  IF fb_RFTrigManualMove.FT THEN
    mManuellMove( bI_Do                  := FALSE
                , fI_TargetPosition      := (fB_Axis.fO_ActualPosition * 1000)
                , fL_ManualMoveTolerance := fB_Axis.fI_Tolerance);
  END_IF
END_IF
(*Rest command if move is done*)
IF bL_Ready OR bL_Error THEN
  sADS_CleanAxis.ResetCommands();
END_IF

sL_CleanDevStatus := sStatus;

(*ADS Feedback*)
sADS_CleanAxis.setFeedback( bManualMoveCanEx := sADS_CleanAxis.bO_ManualMoveCanEx        // do not change
                          , bManualMovekExec := sADS_CleanAxis.bO_ManualMovekExec        // do not change
                          , fAxisPositionVal := fB_Axis.fO_ActualPosition * 1000
                          , wErrorCode       := wL_ErrorCode
                          , bBusy            := sL_CleanDevStatus.bBusy
                          , bReady           := sL_CleanDevStatus.bReady
                          , bError           := sL_CleanDevStatus.bError
                          );


(*----------------------------------------------------------------------------------------------------------------------------------------------- *)
(* Supervision  *)
(*----------------------------------------------------------------------------------------------------------------------------------------------- *)
(*
TODO: Supervisor
tL_TimerSurv.PT := T#3S;
tL_TimerSurv();
tL_TimerSensor.PT := T#105s  ;  (* 1meter at 10mm*)
tL_TimerSensor();*)

IF bL_FirstRun THEN
  bL_FirstRun     := FALSE;
END_IF;

(*----------------------------------------------------------------------------------------------------------------------- *)
(*--------------------------------- Fault Diagnosis and Management  ----------------------------------------------------- *)
(*----------------------------------------------------------------------------------------------------------------------- *)
mErrorHandling();

(*----------------------------------------------------------------------------------------------------------------------- *)
(* Messaging                                                                                                              *)
(*----------------------------------------------------------------------------------------------------------------------- *)
fB_MsgHandler();
fB_Msg[1](bI_Status := bL_Error);
fB_MsgQueue();

METHOD mAckError 
VAR_INPUT
END_VAR
wL_ErrorCode := 0;
mErrorHandling();
fB_Axis.bI_FaultReset := TRUE;
END_METHOD

METHOD mCapping : BOOL
VAR_INPUT
  iI_Step    : INT;
  bI_ExitCap : BOOL;
END_VAR
//Abort: Stop whereever axis is and return
IF bL_AbortReq THEN
  fB_Axis.bI_MoveEnable := FALSE;
  bL_Busy  := FALSE;
  bL_Ready := TRUE;

  RETURN;
END_IF

//Normal operation
bL_Ready := FALSE;
CASE iI_Step OF
	0: //Init - Check if axis is not activated, restore safety
    fB_Axis.bI_MoveEnable := FALSE;
		bL_Busy               := FALSE;

  1: //Wait for PU axis to lift
    mAckError();
    fB_Axis.fI_TargetPosition := (fI_PositionClean1 / 1000);
    fB_Axis.fI_SpeedLimit     := sI_SpeedDef.fP_PlaceSpeed / 1000;
    
    IF bL_InPosClean1 THEN
      fB_Axis.bI_MoveEnable := FALSE;
      bL_Busy               := FALSE;
      bL_Ready              := TRUE;  //Operation complete
    ELSE
      fB_Axis.bI_MoveEnable := bL_SafeMovePos;
      bL_Busy               := TRUE;
    END_IF
    
  2: //Wait for CU axis to move in
    fB_Axis.bI_MoveEnable   := FALSE;
    bL_Busy                 := FALSE;
    
  3: //Move CH to park positiom 
    fB_Axis.bI_MoveEnable   := FALSE;
    bL_Busy                 := FALSE;
    
  4: //Wait for PU axis to lower
    mAckError();
    IF NOT bI_ExitCap THEN
      fB_Axis.fI_TargetPosition := (fI_PositionClean2 / 1000);
      fB_Axis.fI_SpeedLimit     := sI_SpeedDef.fP_PlaceSpeed / 1000;
      
      IF bL_InPosClean2 THEN
        fB_Axis.bI_MoveEnable := FALSE;
        bL_Busy               := FALSE;
        bL_Ready              := TRUE;  //Operation complete
      ELSE
        fB_Axis.bI_MoveEnable := bL_SafeMoveNeg;
        bL_Busy               := TRUE;
      END_IF
    ELSE
      fB_Axis.bI_MoveEnable := FALSE;
      bL_Busy               := FALSE;
    END_IF
    
	5: //End - Do nothing, capping process active
    mAckError();
		bL_Busy  := FALSE;
    bL_Ready := TRUE;  //Operation complete

	ELSE
		bL_Busy  := FALSE;		
    bL_Ready := TRUE;  //Operation complete
END_CASE
END_METHOD

METHOD mCleaning : BOOL
VAR_INPUT
  iI_Step : INT;
END_VAR
//Abort: Stop whereever axis is and return
IF bL_AbortReq THEN
  fB_Axis.bI_MoveEnable := FALSE;
  bL_Busy  := FALSE;
  bL_Ready := TRUE;

  RETURN;
END_IF

//Normal operation
bL_Ready := FALSE;
CASE iI_Step OF
  0: //Init - Check if axis is not activated, restore safety
    bL_Busy := FALSE;

  1: //Wait for PU axis to lift
    mAckError();
    fB_Axis.fI_TargetPosition := (fI_PositionClean1 / 1000);
    fB_Axis.fI_SpeedLimit     := sI_SpeedDef.fP_PlaceSpeed / 1000;
    
    IF bL_InPosClean1 THEN
      fB_Axis.bI_MoveEnable := FALSE;
      bL_Busy               := FALSE;
      bL_Ready              := TRUE;  //Operation complete
    ELSE
      fB_Axis.bI_MoveEnable := bL_SafeMovePos;
      bL_Busy               := TRUE;
    END_IF
    
  2: //Wait for CU axis to move in
    fB_Axis.bI_MoveEnable   := FALSE;
    bL_Busy                 := FALSE;
    
  3: //Wait for PU axis to lower
    mAckError();
    fB_Axis.fI_TargetPosition := (fI_PositionClean2 / 1000);
    fB_Axis.fI_SpeedLimit     := sI_SpeedDef.fP_PlaceSpeed / 1000;
    
    IF bL_InPosClean2 THEN
      fB_Axis.bI_MoveEnable := FALSE;
      bL_Busy               := FALSE;
      bL_Ready              := TRUE;  //Operation complete
    ELSE
      fB_Axis.bI_MoveEnable := bL_SafeMoveNeg;
      bL_Busy               := TRUE;
    END_IF
    
  4: //Ensure CH axis is at starting position
    fB_Axis.bI_MoveEnable   := FALSE;
    bL_Busy                 := FALSE;
    
  5: //Move CH to clean start position
    fB_Axis.bI_MoveEnable   := FALSE;
    bL_Busy                 := FALSE;

  6: //Wait until cleaning equipment ready
    fB_Axis.bI_MoveEnable   := FALSE;
    bL_Busy                 := FALSE;
    
  7: //Cleaning
    fB_Axis.bI_MoveEnable   := FALSE;
    bL_Busy                 := FALSE;  
    
  8: //Wait until cleaning equipment ready
    fB_Axis.bI_MoveEnable   := FALSE;
    bL_Busy                 := FALSE;
    
  9: //Move CH to end position
    fB_Axis.bI_MoveEnable   := FALSE;
    bL_Busy                 := FALSE;  
    
  10: //Wait for PU axis to lift
    mAckError();
    fB_Axis.fI_TargetPosition := (fI_PositionClean1 / 1000);
    fB_Axis.fI_SpeedLimit     := sI_SpeedDef.fP_PlaceSpeed / 1000;
    
    IF bL_InPosClean1 THEN
      fB_Axis.bI_MoveEnable := FALSE;
      bL_Busy               := FALSE;
      bL_Ready              := TRUE;  //Operation complete
    ELSE
      fB_Axis.bI_MoveEnable := bL_SafeMovePos;
      bL_Busy               := TRUE;
    END_IF
  
  11: //Move CH back to start 
    fB_Axis.bI_MoveEnable   := FALSE;
    bL_Busy                 := FALSE;  

  12: //Wait for PU axis to lower
    mAckError();
    fB_Axis.fI_TargetPosition := (fI_PositionClean2 / 1000);
    fB_Axis.fI_SpeedLimit     := sI_SpeedDef.fP_PlaceSpeed / 1000;
    
    IF bL_InPosClean2 THEN
      fB_Axis.bI_MoveEnable := FALSE;
      bL_Busy               := FALSE;
      bL_Ready              := TRUE;  //Operation complete
    ELSE
      fB_Axis.bI_MoveEnable := bL_SafeMoveNeg;
      bL_Busy               := TRUE;
    END_IF
    
  13: //End
    fB_Axis.bI_MoveEnable   := FALSE;
    bL_Busy                 := FALSE;  
    bL_Ready                := TRUE;  //Operation complete
  
  ELSE
    bL_Busy  := FALSE;    
    bL_Ready := TRUE;  //Operation complete
END_CASE
END_METHOD

METHOD PRIVATE mErrorHandling
VAR_INPUT
END_VAR
fB_Msg[1].bI_Status := FALSE;

IF NOT bL_RefKnown THEN
	wL_ErrorCode.1 := TRUE;						(* Axis has lost its value *)
END_IF;

IF (NOT bI_SensorTop AND NOT bI_SensorBottom) THEN      (* Sensor Fault : SensorTop and SensorBottom can't be active at the same time *)
	wL_ErrorCode.2 := TRUE;
END_IF;

IF (NOT bI_SensorTop AND bL_MemSensorTop) THEN          (* Safety Fault : Limit Switch Top activated *)
	wL_ErrorCode.3 := TRUE;
END_IF;
bL_MemSensorTop := bI_SensorTop;

IF (NOT bI_SensorBottom AND bL_MemSensorBottom) THEN    (* Safety Fault : Limit Switch Bottom activated *)
	wL_ErrorCode.4 := TRUE;
END_IF;
bL_MemSensorBottom := bI_SensorBottom;

IF (sI_SpeedDef.fP_PlaceSpeed=0) OR  (sI_SpeedDef.fP_WorkSpeed=0) OR (sI_SpeedDef.fP_ServiceSpeed=0) THEN	(* Speed Configuration not done *)
	wL_Errorcode.6 := TRUE;
END_IF;

IF (fI_PositionService = 0) OR (fI_PositionWait = 0) OR (fI_PositionClean1 = 0) OR (fI_PositionClean2 = 0) THEN		(* Position Configuration not done *)
	wL_ErrorCode.7 := TRUE;
END_IF;

IF fB_Axis.eO_EL7201Status = eFault  THEN
	wL_ErrorCode.8 := TRUE;						(* EL7342 module fault *)
	fB_Msg[1].bI_Status := TRUE;
END_IF;


IF wl_ErrorCode = 0 THEN
	bL_Error := FALSE;
ELSE
	bL_Error := TRUE;
END_IF;
END_METHOD

METHOD mErrorRecovery : BOOL
VAR_INPUT
    iI_Step : INT;
END_VAR
//Do nothing
bL_Busy  := FALSE;
bL_Ready := TRUE;
END_METHOD

METHOD mInit
VAR_INPUT
END_VAR
	(*Messages*)
	sL_MsgConfig.bI_Enable       := TRUE;
	sL_MsgConfig.pI_FbMsgHandler := ADR(fB_MsgHandler);
	fB_MsgHandler.pI_MsgQueue    := ADR(fB_MsgQueue);
	fB_MsgQueue.pI_MsgInterface  := ADR(sADS_CleanAxis.sO_Message);
	fB_MsgQueue.cI_MaxElement    := 5;

	fB_Msg[1].iI_MsgLocation     := TO_INT(eMa_BLK_CLEANAXIS);
	fB_Msg[1].pI_MsgConfig       := ADR(sL_MsgConfig);
	fB_Msg[1].iI_MsgNumber       := eCMa_AxisErrorZ;
END_METHOD

METHOD mManuellMove : BOOL
VAR_INPUT
  bI_Do                  : BOOL;
  fI_TargetPosition      : REAL;
  fL_ManualMoveTolerance : REAL;
END_VAR
IF fB_Axis.fO_ActualPosition < (fI_PositionWait / 1000) THEN
  fB_Axis.fI_SpeedLimit   := sI_SpeedDef.fP_WorkSpeed / 1000;
ELSE
  fB_Axis.fI_SpeedLimit   := sI_SpeedDef.fP_ServiceSpeed / 1000;
END_IF
fB_Axis.fI_TargetPosition := fI_TargetPosition / 1000;
IF fB_Axis.fI_TargetPosition > fB_Axis.fO_ActualPosition THEN
  fB_Axis.bI_MoveEnable   := bI_Do AND bL_SafeMovePos;
ELSIF fB_Axis.fI_TargetPosition < fB_Axis.fO_ActualPosition THEN
  fB_Axis.bI_MoveEnable   := bI_Do AND bL_SafeMoveNeg;
ELSE
  fB_Axis.bI_MoveEnable   := bI_Do;
END_IF

bL_Busy  := ABS(fB_Axis.fI_TargetPosition - fB_Axis.fO_ActualPosition) > fL_ManualMoveTolerance;
bL_Ready := NOT (ABS(fB_Axis.fI_TargetPosition - fB_Axis.fO_ActualPosition) > fL_ManualMoveTolerance);  //Operation complete
END_METHOD

METHOD mPrintPos : BOOL
VAR_INPUT
  bI_PrintEnabled        : BOOL;
  bI_PrintFinsihed       : BOOL;
END_VAR

VAR
  bDriveToWaitPos        : BOOL;
  bDriveToPrintPos       : BOOL;
END_VAR
fb_RFTrigPrintEnabled(CLK := bI_PrintEnabled);
IF fb_RFTrigPrintEnabled.RT THEN bL_DriveToPrintPos := TRUE; bL_DriveToWaitPos  := FALSE; END_IF
IF fb_RFTrigPrintEnabled.FT THEN bL_DriveToWaitPos  := TRUE; bL_DriveToPrintPos := FALSE; END_IF

IF NOT pHigherPosWait AND bL_Ready THEN
  //IF fb_RFTrigPrintEnabled.RT THEN bL_DriveToPrintPos := TRUE; END_IF
  IF bL_DriveToPrintPos THEN
    fB_Axis.fI_TargetPosition := (fL_PrintPosition);
    fB_Axis.fI_SpeedLimit     := sI_SpeedDef.fP_WorkSpeed / 1000;
    
    IF bL_InPosPrint THEN
      fB_Axis.bI_MoveEnable := FALSE;
      bL_Busy               := FALSE;
      bL_DriveToPrintPos    := FALSE;
      bL_Ready              := TRUE;  //Operation complete
    ELSE
      fB_Axis.bI_MoveEnable := bL_SafeMoveNeg;
      bL_Busy               := TRUE;
    END_IF
  END_IF

  //IF fb_RFTrigPrintEnabled.FT THEN bL_bDriveToWaitPos := TRUE; END_IF
  IF bL_DriveToWaitPos AND bI_PrintFinsihed THEN
    fB_Axis.fI_TargetPosition := (fI_PositionWait / 1000);
    fB_Axis.fI_SpeedLimit     := sI_SpeedDef.fP_PlaceSpeed / 1000;
    
    IF bL_InPosWait THEN
      fB_Axis.bI_MoveEnable := FALSE;
      bL_Busy               := FALSE;
      bL_DriveToWaitPos     := FALSE;
      bL_Ready              := TRUE;  //Operation complete
    ELSE
      fB_Axis.bI_MoveEnable := bL_SafeMovePos;
      bL_Busy               := TRUE;
    END_IF
  END_IF
END_IF
END_METHOD

METHOD mProduction : BOOL
VAR_INPUT
  iI_Step : INT;
END_VAR
//Abort: Stop whereever axis is and return
IF bL_AbortReq THEN
  fB_Axis.bI_MoveEnable := FALSE;
  bL_Busy  := FALSE;
  bL_Ready := TRUE;

  RETURN;
END_IF

//Normal operation
bL_Ready := FALSE;
CASE iI_Step OF
  0: //Init - Check if axis is not activated, restore safety
    bL_Busy := FALSE;

  1: //Wait for PU axis to lift
    mAckError();
    fB_Axis.fI_TargetPosition := (fI_PositionClean1 / 1000);
    fB_Axis.fI_SpeedLimit     := sI_SpeedDef.fP_PlaceSpeed / 1000;
    
    IF bL_InPosClean1 THEN
      fB_Axis.bI_MoveEnable := FALSE;
      bL_Busy               := FALSE;
      bL_Ready              := TRUE;  //Operation complete
    ELSE
      fB_Axis.bI_MoveEnable := bL_SafeMovePos;
      bL_Busy               := TRUE;
    END_IF
    
  2: //Wait for CU axis to move out
    fB_Axis.bI_MoveEnable   := FALSE;
    bL_Busy                 := FALSE;
    
  3: //Wait for PU axis to lower
    mAckError();
    fB_Axis.fI_TargetPosition := (fI_PositionWait / 1000);
    fB_Axis.fI_SpeedLimit     := sI_SpeedDef.fP_PlaceSpeed / 1000;
    
    IF bL_InPosWait THEN
      fB_Axis.bI_MoveEnable := FALSE;
      bL_Busy               := FALSE;
      bL_Ready              := TRUE;  //Operation complete
    ELSE
      fB_Axis.bI_MoveEnable := bL_SafeMoveNeg;
      bL_Busy               := TRUE;
    END_IF
    
  4: //End
    fB_Axis.bI_MoveEnable := FALSE;
    bL_Busy               := FALSE;  
    bL_Ready              := TRUE;  //Operation complete

  ELSE
    bL_Busy  := FALSE;    
    bL_Ready := TRUE;  //Operation complete
END_CASE
END_METHOD

METHOD mService : BOOL
VAR_INPUT
  iI_Step : INT;
END_VAR
//Abort: Stop whereever axis is and return
IF bL_AbortReq THEN
  fB_Axis.bI_MoveEnable := FALSE;
  bL_Busy  := FALSE;
  bL_Ready := TRUE;

  RETURN;
END_IF

//Normal operation
bL_Ready := FALSE;
CASE iI_Step OF
  0: //Init - Check if axis is not activated, restore safety
    bL_Busy := FALSE;

  1: //Wait for PU axis to lift to ExitCapping
    mAckError();
    fB_Axis.fI_TargetPosition := (fI_PositionClean1 / 1000);
    fB_Axis.fI_SpeedLimit     := sI_SpeedDef.fP_PlaceSpeed / 1000;
    
    IF bL_InPosClean1 THEN
      fB_Axis.bI_MoveEnable := FALSE;
      bL_Busy               := FALSE;
    ELSE
      fB_Axis.bI_MoveEnable := bL_SafeMovePos;
      bL_Busy               := TRUE;
    END_IF
        
  2: //Wait for PU to reach Service (CU moves out)
    mAckError();
    fB_Axis.fI_TargetPosition := (fI_PositionService / 1000);
    fB_Axis.fI_SpeedLimit     := sI_SpeedDef.fP_PlaceSpeed / 1000;
    
    IF bL_InPosService THEN
      fB_Axis.bI_MoveEnable := FALSE;
      bL_Busy               := FALSE;
      bL_Ready              := TRUE;  //Operation complete
    ELSE
      fB_Axis.bI_MoveEnable := bL_SafeMovePos;
      bL_Busy               := TRUE;
    END_IF
    
  3: //End
    fB_Axis.bI_MoveEnable := FALSE;
    bL_Busy               := FALSE; 
    bL_Ready              := TRUE; 
  
  ELSE
    bL_Busy  := FALSE;    
    bL_Ready := TRUE;  //Operation complete
END_CASE
END_METHOD

METHOD mStartup : BOOL
VAR_INPUT
  iI_Step : INT;
END_VAR
CASE iI_Step OF
	0: //Init - Check if axis is not activated, restore safety
		bL_Busy := FALSE;

  1: //Wait for PU axis to lift
    mAckError();
    fB_Axis.fI_TargetPosition := (fI_PositionClean1 / 1000);
    fB_Axis.fI_SpeedLimit     := sI_SpeedDef.fP_PlaceSpeed / 1000;
    
    IF bL_InPosClean1 OR bL_HigherPosC1 THEN
      fB_Axis.bI_MoveEnable := FALSE;
      bL_Busy               := FALSE;
      bL_Ready              := TRUE;  //Operation complete
    ELSE
      fB_Axis.bI_MoveEnable := bL_SafeMovePos;
      bL_Busy               := TRUE;
    END_IF
    
	2,3,4: //End
		bL_Busy  := FALSE;		
    bL_Ready := TRUE;  //Operation complete

	ELSE
		bL_Busy  := FALSE;		
    bL_Ready := TRUE;  //Operation complete
END_CASE
END_METHOD

{attribute 'monitoring' := 'call'}
PROPERTY pHigherPosC1 : bool
GET
pHigherPosC1 := bL_HigherPosC1;
END_GET
END_PROPERTY

{attribute 'monitoring' := 'call'}
PROPERTY pHigherPosWait : bool
GET
pHigherPosWait := bL_HigherPosWait;
END_GET
END_PROPERTY

{attribute 'monitoring' := 'call'}
PROPERTY pInPosClean1 : bool
GET
pInPosClean1 := bL_InPosClean1;
END_GET
END_PROPERTY

{attribute 'monitoring' := 'call'}
PROPERTY pInPosClean2 : bool
GET
pInPosClean2 := bL_InPosClean2;
END_GET
END_PROPERTY

{attribute 'monitoring' := 'call'}
PROPERTY pInPosPrint : bool
GET
pInPosPrint := bL_InPosPrint;
END_GET
END_PROPERTY

{attribute 'monitoring' := 'call'}
PROPERTY pInPosService : bool
GET
pInPosService := bL_InPosService;
END_GET
END_PROPERTY

{attribute 'monitoring' := 'call'}
PROPERTY pInPosWait : bool
GET
pInPosWait := bL_InPosWait;
END_GET
END_PROPERTY

PROPERTY pPositionPrint : REAL
GET
pPositionPrint := fI_PositionPrint;
END_GET
SET
fI_PositionPrint := pPositionPrint;
END_SET
END_PROPERTY

PROPERTY setPlaceSpeed : REAL
SET
sI_SpeedDef.fP_PlaceSpeed := setPlaceSpeed;
END_SET
END_PROPERTY

END_FUNCTION_BLOCK

// ---- POUs/Machine/CleaningStation/FB_CleaningProcess.TcPOU
FUNCTION_BLOCK FB_CleaningProcess EXTENDS FB_MachineBase IMPLEMENTS I_CleaningStateCallback
VAR_INPUT
  I_CleanDeviceList              : ARRAY[1..cI_MAXCLEANDEVICES] OF I_CleanDevice;

  (*User commands*)
  bI_UsrService                  : BOOL;                         (*User has selected service (1) or print(0) mode*)
  bI_UsrAbort                    : BOOL;                         (*User aborted*)
  bI_Emergency                   : BOOL;
  bI_SafetyOk                    : BOOL;

  bI_CappingCommand              : BOOL;                         (*Capping command*)
  bI_PurgeCommand                : BOOL;                         (*Purge command*)
  bI_CleanCommand                : BOOL;                         (*Clean command*)
  bI_CleanLocked                 : BOOL;                         (*Cleaning locked*)
  
  (*User settings*)
  bI_UsrAutoMode                 : BOOL;                         (*User has selected automatic mode*)
  bI_UsrCleanAfterPurge          : BOOL;                         (*Automatically clean after Purge*)
  bI_UsrCleanAfterCapp           : BOOL;                         (*Automatically clean after Capping*)
  bI_UsrPurgeAfterCapp           : BOOL;                         (*Automatically purge after Capping*)

  bI_CappingPosReached           : BOOL;                         (*Capping position reached*)
  bI_CappingEnterPosReached      : BOOL;                         (*Capping enter position reached*)
END_VAR

VAR_OUTPUT
END_VAR

VAR
  sADS_CleanProcess              : FB_ADS_CleanProcess;

  fB_StateInit                   : FB_CleaningProcessStateInit;
  fB_StateProduction             : FB_CleaningProcessStateProduction;
  fB_StateService                : FB_CleaningProcessStateService;
  fB_StateCapping                : FB_CleaningProcessStateCapping;
  fB_StateCappingExit            : FB_CleaningProcessStateCappingExit;
  fB_StateCleaning               : FB_CleaningProcessStateCleaning;
  fB_StateError                  : FB_CleaningProcessStateError;
  sL_CurrentState                : POINTER TO FB_CleaningProcessStateBase;
  
  bL_UsrService                  : BOOL;
  bL_UsrProductionRequest        : BOOL;
  bL_UsrServiceRequest           : BOOL;
  bL_Abort                       : BOOL;  
  bL_AbortExec                   : BOOL;
  sL_DeviceStatus                : ST_CLEANING_DEV_STATUS;

  bL_PurgeExec                   : BOOL;
  
  iL_CleanDeviceCount            : INT;
  iL_CdCount                     : INT;
END_VAR

VAR CONSTANT
  cI_MAXCLEANDEVICES             : INT := 10;
END_VAR

//Current state cyclic action
sL_CurrentState^.mStateAction();

IF sL_CurrentState^.pInitDone THEN
  IF bI_UsrService AND NOT bL_UsrService THEN //Switch to service
    bL_UsrServiceRequest    := TRUE;
    bL_UsrProductionRequest := FALSE;
  ELSIF NOT bI_UsrService AND bL_UsrService THEN //Switch to production
    bL_UsrProductionRequest := TRUE;
    bL_UsrServiceRequest    := FALSE;
  END_IF
  
  bL_UsrService := bI_UsrService;
END_IF
  
//Decode user commands
mUserCommand();

//Get device status
sL_DeviceStatus := mDeviceStatus();

METHOD mAckError : BOOL
VAR_INPUT
END_VAR
mDeviceAckError();

//Get device status
sL_DeviceStatus := mDeviceStatus();

IF bI_UsrAutoMode THEN
  sL_CurrentState^.mAckError();
END_IF

sADS_CleanProcess.bAcknowledgeError := FALSE;
END_METHOD

METHOD mChangeState
VAR_INPUT
	sI_NextState	: EN_Cleaning_State;
END_VAR

VAR
  	sL_PrevState	: POINTER TO FB_CleaningProcessStateBase;
END_VAR
//Exit action
sL_CurrentState^.mExitAction();

//Switch state
sL_PrevState:=sL_CurrentState;

CASE sI_NextState OF
	EN_Cleaning_State.Init:
		sL_CurrentState:=ADR(fB_StateInit);
	EN_Cleaning_State.Production:
		sL_CurrentState:=ADR(fB_StateProduction);
	EN_Cleaning_State.Service:
		sL_CurrentState:=ADR(fB_StateService);
	EN_Cleaning_State.Capping:
		sL_CurrentState:=ADR(fB_StateCapping);
	EN_Cleaning_State.CappingExit:
		sL_CurrentState:=ADR(fB_StateCappingExit);
	EN_Cleaning_State.Cleaning:
		sL_CurrentState:=ADR(fB_StateCleaning);
	EN_Cleaning_State.Error:
		sL_CurrentState:=ADR(fB_StateError);	
END_CASE

//Entry action
sL_CurrentState^.mEntryAction();
END_METHOD

METHOD mDeviceAbort : BOOL

VAR
  bL_Success       : BOOL;
END_VAR
bL_Success := TRUE;

//Populate command
FOR iL_CdCount := 1 TO iL_CleanDeviceCount DO
	bL_Success := bL_Success AND I_CleanDeviceList[iL_CdCount].mAbort();
END_FOR

mDeviceAbort:=TRUE;
END_METHOD

METHOD mDeviceAckError
VAR_INPUT
END_VAR
//Populate command
FOR iL_CdCount := 1 TO iL_CleanDeviceCount DO
	I_CleanDeviceList[iL_CdCount].mAckError();
END_FOR
END_METHOD

METHOD mDeviceOperation : BOOL
VAR_INPUT
  iI_Step    : INT;	
END_VAR

VAR
  bL_Success : BOOL;
END_VAR
bL_Success := TRUE;

//Populate command
FOR iL_CdCount := 1 TO iL_CleanDeviceCount DO
	bL_Success := bL_Success AND I_CleanDeviceList[iL_CdCount].mOperation(iI_Step);
END_FOR

//Return result
mDeviceOperation := bL_Success;
END_METHOD

METHOD PROTECTED mDeviceStatus : ST_CLEANING_DEV_STATUS
VAR
  sL_GlobalStatus : ST_CLEANING_DEV_STATUS;
  sL_DeviceStatus : ST_CLEANING_DEV_STATUS;
END_VAR
sL_GlobalStatus.bBusy     := FALSE;
sL_GlobalStatus.bError    := FALSE;
sL_GlobalStatus.bReady    := TRUE;
sL_GlobalStatus.bRefKnown := TRUE;

//Get status
FOR iL_CdCount := 1 TO iL_CleanDeviceCount DO
	sL_DeviceStatus := I_CleanDeviceList[iL_CdCount].sStatus;
	
	sL_GlobalStatus.bBusy     := sL_GlobalStatus.bBusy      OR sL_DeviceStatus.bBusy;
	sL_GlobalStatus.bError    := sL_GlobalStatus.bError     OR sL_DeviceStatus.bError;
	sL_GlobalStatus.bReady    := sL_GlobalStatus.bReady    AND sL_DeviceStatus.bReady;
	sL_GlobalStatus.bRefKnown := sL_GlobalStatus.bRefKnown AND sL_DeviceStatus.bRefKnown;
END_FOR

//Return result
mDeviceStatus := sL_GlobalStatus;
END_METHOD

METHOD PUBLIC mInit : BOOL
VAR_INPUT
	
END_VAR
//Init states
fB_StateInit       .mInit(I_MachineStatus, THIS^);		
fB_StateProduction .mInit(I_MachineStatus, THIS^);	 
fB_StateService    .mInit(I_MachineStatus, THIS^);	 	
fB_StateCapping    .mInit(I_MachineStatus, THIS^);	 	
fB_StateCappingExit.mInit(I_MachineStatus, THIS^);	 	
fB_StateCleaning   .mInit(I_MachineStatus, THIS^);	 	
fB_StateError      .mInit(I_MachineStatus, THIS^);	 		

//State names
fB_StateInit       .pName := 'Init';
fB_StateProduction .pName := 'Production';
fB_StateService    .pName := 'Service';
fB_StateCapping    .pName := 'CappingEnter';
fB_StateCappingExit.pName := 'CappingExit';
fB_StateCleaning   .pName := 'Cleaning';
fB_StateError      .pName := 'Error';

//Set initial state
sL_CurrentState := ADR(fB_StateInit);
END_METHOD

METHOD PUBLIC mRegisterDevice : BOOL
VAR_INPUT
  I_NewDevice : I_CleanDevice;
END_VAR
IF iL_CleanDeviceCount < cI_MAXCLEANDEVICES AND I_NewDevice <> 0 THEN
  iL_CleanDeviceCount := iL_CleanDeviceCount + 1;
  I_CleanDeviceList[iL_CleanDeviceCount] := I_NewDevice;
END_IF
END_METHOD

METHOD mSetMode : BOOL
VAR_INPUT
  sI_CleanMode     : EN_CLEANING_OP;
END_VAR

VAR
  bL_Success       : BOOL;
END_VAR
bL_Success := TRUE;

//Populate command
FOR iL_CdCount := 1 TO iL_CleanDeviceCount DO
	bL_Success := bL_Success AND I_CleanDeviceList[iL_CdCount].mSetMode(sI_CleanMode);
END_FOR

//Return result
mSetMode := bL_Success;
END_METHOD

METHOD mUserCommand
VAR_INPUT
END_VAR

VAR
	bL_ServiceResult     : BOOL;
  bL_CleanProcessCanEx : BOOL;
END_VAR
(*Abort command*)
IF    ((bI_UsrAbort OR sADS_CleanProcess.bI_Abort) AND NOT bL_Abort)  //Rising edge of abort command
   OR NOT I_MachineStatus.pSafetyOk
THEN
  bL_Abort             := TRUE;
  bL_AbortExec         := TRUE;
  bL_ServiceResult     := sL_CurrentState^.mAbort();

  (*Reset commands*)
  bL_UsrProductionRequest := FALSE;
  bL_UsrServiceRequest    := FALSE;
  sADS_CleanProcess.ResetCommands();
ELSE
  IF NOT (bI_UsrAbort OR sADS_CleanProcess.bI_Abort) THEN
    bL_Abort           := FALSE;
  END_IF
  bL_AbortExec         := FALSE;
END_IF

  
(*Select Operation*) 
IF bI_UsrAutoMode THEN
  IF sADS_CleanProcess.bI_Maintenance THEN
    bL_ServiceResult := sL_CurrentState^.mService();
  ELSIF bL_UsrProductionRequest THEN
    bL_ServiceResult := sL_CurrentState^.mProduction();
    IF bL_ServiceResult THEN
      bL_UsrProductionRequest := FALSE;
    END_IF
  ELSIF (bI_CappingCommand OR sADS_CleanProcess.bI_StartCapping OR bL_UsrServiceRequest) AND NOT bI_CappingEnterPosReached THEN
    bL_ServiceResult := sL_CurrentState^.mCleaningOp(EN_CLEANING_OP.eOPCAPENTER);
    IF bL_ServiceResult THEN
      bL_UsrServiceRequest := FALSE;
    END_IF
  ELSIF sADS_CleanProcess.bI_StopCapping THEN
    bL_ServiceResult := sL_CurrentState^.mCleaningOp(EN_CLEANING_OP.eOPCAPEXIT);
  ELSIF (bI_CleanCommand OR sADS_CleanProcess.bI_Clean) AND NOT bI_CleanLocked THEN
    bL_ServiceResult := sL_CurrentState^.mCleaningOp(EN_CLEANING_OP.eOPCLEAN);
  (*
  ELSIF sADS_CleanProcess.bI_Maintenance THEN
    bL_ServiceResult := sL_CurrentState^.mCleaningOp(EN_CLEANING_OP.eOPMAINT);
  *)
  ELSIF (bI_PurgeCommand OR sADS_CleanProcess.bI_Purge) AND NOT bI_CleanLocked THEN
    bL_PurgeExec := TRUE;
    IF NOT bI_CappingPosReached THEN
      bL_ServiceResult := sL_CurrentState^.mCleaningOp(EN_CLEANING_OP.eOPPURGE);
    END_IF
  (*
  ELSIF sADS_CleanProcess.bI_OpenShutter THEN
    bL_ServiceResult := sL_CurrentState^.mCleaningOp(EN_CLEANING_OP.eOPSHUTTEROPEN);
  *)
  END_IF
END_IF

//Error handling
IF NOT bL_ServiceResult THEN
	; //TODO Implement error message
END_IF

//ACK Error from cleaning GUI
IF sADS_CleanProcess.bI_AcknowledgeError THEN
  mAckError();
END_IF

//Command handshake
//TODO: HANDLE PURGE CanEx Ex properly

bL_CleanProcessCanEx := bI_UsrAutoMode  AND bI_UsrService AND NOT sL_DeviceStatus.bBusy;

sADS_CleanProcess.setFeedback( bStartCappingCanEx       := bL_CleanProcessCanEx
                             , bStartCappingExec        := fB_StateCapping.bL_DevOpActive
          
                             , bStopCappingCanEx        := bL_CleanProcessCanEx
                             , bStopCappingExec         := fB_StateCappingExit.bL_DevOpActive
          
                             , bPurgeCanEx              := bL_CleanProcessCanEx
                             , bPurgeExec               := bL_PurgeExec
          
                             , bCleanCanEx              := bL_CleanProcessCanEx AND NOT bI_CleanLocked
                             , bCleanExec               := fB_StateCleaning.bL_DevOpActive
          
                             , bMaintenanceCanEx        := bL_CleanProcessCanEx
                             , bMaintenanceExec         := fB_StateService.bL_DevOpActive
          
                             , bOpenShutterCanEx        := FALSE  (*DEM: not exists*)
                             , bOpenShutterExec         := FALSE  (*DEM: not exists*)
          
                             , bAbortCanEx              := sL_DeviceStatus.bBusy OR sL_DeviceStatus.bError
                             , bAbortExec               := bL_AbortExec
          
                             , bAcknowledgeErrorCanEx   := sL_DeviceStatus.bError OR NOT sL_DeviceStatus.bRefKnown OR (sL_CurrentState^.sL_StateName = fB_StateError.pName)
                             , bAcknowledgeErrorExec    := FALSE
          
                             , bBusy                    := sL_DeviceStatus.bBusy
                             , bReady                   := TRUE
                             , bServiceEnabled          := FALSE
                             , bAxisProcessMovingVisible:= TRUE
          
                             , wErrorCode               := 0
                             );
END_METHOD

PROPERTY pDeviceStatus : ST_CLEANING_DEV_STATUS
GET
pDeviceStatus := sL_DeviceStatus;
END_GET
END_PROPERTY

PROPERTY pPurgeExec : BOOL
GET
pPurgeExec := bL_PurgeExec;
END_GET
SET
bL_PurgeExec := pPurgeExec;
END_SET
END_PROPERTY

END_FUNCTION_BLOCK

// ---- POUs/Machine/CleaningStation/FB_CleaningProcessStateInit.TcPOU
FUNCTION_BLOCK FB_CleaningProcessStateInit EXTENDS FB_CleaningProcessStateBase
VAR_INPUT
END_VAR
VAR_OUTPUT
END_VAR
VAR
	bL_InitActive : BOOL := TRUE;;
END_VAR

METHOD mProduction : BOOL
VAR_INPUT
END_VAR
//Switch to production mode if no operation active
IF I_MachineStatus.pSafetyOk AND I_MachineStatus.pMachineReady AND NOT bL_DevOpActive THEN
	I_ParentCallback.mChangeState(EN_Cleaning_State.Production);
END_IF
END_METHOD

METHOD mService : BOOL
VAR_INPUT
END_VAR
//Switch to service mode
IF NOT bL_DevOpActive THEN
	I_ParentCallback.mChangeState(EN_Cleaning_State.Service);
END_IF
END_METHOD

METHOD mStateAction
VAR_INPUT
END_VAR

VAR
	sL_DeviceStatus : ST_CLEANING_DEV_STATUS;
END_VAR
sL_DeviceStatus := I_ParentCallback.pDeviceStatus;

//If safety ok try to reference axes
IF I_MachineStatus.pSafetyOk AND I_MachineStatus.pMachineReady AND NOT bL_DevOpActive THEN
	//Set mode and start process when successful
	bL_DevOpActive := I_ParentCallback.mSetMode(EN_CLEANING_OP.eOPSTARTUP);
END_IF

IF bL_DevOpActive THEN
	mDevOp();	
END_IF

//If all axes referenced go to service mode
IF sL_DeviceStatus.bError THEN
	I_ParentCallback.mChangeState(EN_Cleaning_State.Error);
ELSIF sL_DeviceStatus.bRefKnown AND NOT sL_DeviceStatus.bBusy THEN
	//I_ParentCallback.mChangeState(EN_Cleaning_State.Service);
	I_ParentCallback.mChangeState(EN_Cleaning_State.Capping);

  bL_InitActive    := FALSE;
  SUPER^.pInitDone := TRUE;
END_IF
END_METHOD

PROPERTY pInitDone : BOOL
GET
pInitDone := NOT bL_InitActive;
END_GET
END_PROPERTY

END_FUNCTION_BLOCK

// ---- POUs/Machine/CleaningStation/FB_CleaningProcessStateBase.TcPOU
FUNCTION_BLOCK FB_CleaningProcessStateBase
VAR_INPUT
  I_ParentCallback : I_CleaningStateCallback;
  I_MachineStatus  : I_MachineStateBase;
END_VAR

VAR_OUTPUT
END_VAR

VAR
  sL_StateName	 : STRING;
	
  //Device operation
  iL_CurrentStep : INT;
  iL_State       : INT := 1;
  bL_DevOpActive : BOOL;
  bL_AbortPend   : BOOL;
END_VAR

VAR_STAT
  bL_InitDone    : BOOL := FALSE;
END_VAR	

VAR CONSTANT
  //Device operation
  cL_SEND    : INT := 1;
  cL_WAIT    : INT := 2;	
  cL_NEXT    : INT := 3;	
  cL_DONE    : INT := 4;
  cL_ERROR   : INT := 5;

  cL_MaxStep : INT := 15; //Make dynamic one day	
END_VAR

//No code here, use mStateAction

METHOD mAbort : BOOL
VAR_INPUT
END_VAR
IF NOT bL_AbortPend THEN
  I_ParentCallback.mDeviceAbort();
  bL_AbortPend:=TRUE;
  
  IF NOT bL_DevOpActive THEN
    bL_DevOpActive := TRUE; //Set to relaunch process
    iL_CurrentStep := 0;
	END_IF
END_IF
END_METHOD

METHOD mAckError : BOOL
VAR_INPUT
END_VAR
END_METHOD

METHOD mCleaningOp : BOOL
VAR_INPUT
	sI_Operation : EN_CLEANING_OP;
END_VAR
//Service not implemented
mCleaningOp:=FALSE;
END_METHOD

METHOD mDevOp
VAR_INPUT
END_VAR

VAR
  sL_Status : ST_CLEANING_DEV_STATUS;
END_VAR
sL_Status := I_ParentCallback.pDeviceStatus;
I_ParentCallback.mDeviceOperation(iL_CurrentStep);

CASE iL_State OF
  // Send command to devices
  cL_SEND:
    iL_State := cL_WAIT;  
    
  // Wait until operation completed  
  cL_WAIT:
    IF sL_Status.bError THEN
      iL_State := cL_ERROR;
    ELSIF NOT sL_Status.bBusy THEN
      iL_State := cL_NEXT;
    END_IF
    
  // Next state 
  cL_NEXT:
    IF iL_CurrentStep < cL_MaxStep AND NOT sL_Status.bReady THEN
      iL_CurrentStep := iL_CurrentStep + 1;  

      iL_State := cL_SEND;
    ELSE
      iL_State := cL_DONE;
    END_IF
    
  // Done
  cL_DONE:
    bL_DevOpActive := FALSE; //Clear cleaning flag
    iL_State       := cL_SEND; //Init for next operation
    iL_CurrentStep := 0;
    I_ParentCallback.mSetMode(EN_CLEANING_OP.eNOP);
    mDevOpDone();
  
  // Error
  cL_ERROR:
    bL_DevOpActive := FALSE; //Clear cleaning flag
    iL_State       := cL_SEND; //Init for next operation
    iL_CurrentStep := 0;
END_CASE
END_METHOD

METHOD mDevOpDone : BOOL
VAR_INPUT
END_VAR
//Optional action when device operation completed

//Operation (incl. Abort) terminated
bL_AbortPend:=FALSE;
END_METHOD

METHOD mEntryAction
VAR_INPUT
END_VAR
END_METHOD

METHOD mExitAction
VAR_INPUT
END_VAR
END_METHOD

METHOD mInit : BOOL
VAR_INPUT
  I_parentMachineState : I_MachineStateBase;
  I_Callback           : I_CleaningStateCallback;
END_VAR
I_MachineStatus  := I_parentMachineState;
I_ParentCallback := I_Callback;
END_METHOD

METHOD mProduction : BOOL
VAR_INPUT
END_VAR
//Request production mode - implement in SubClass
mProduction := FALSE;
END_METHOD

METHOD mService : BOOL
VAR_INPUT
END_VAR
//Request service mode - implement in SubClass
mService := FALSE;
END_METHOD

METHOD mStateAction
VAR_INPUT
END_VAR

VAR
	sL_DeviceStatus: ST_CLEANING_DEV_STATUS;
END_VAR
sL_DeviceStatus := I_ParentCallback.pDeviceStatus;

//If a device has an error go to error state
IF sL_DeviceStatus.bError THEN
	I_ParentCallback.mChangeState(EN_Cleaning_State.Error);
END_IF
END_METHOD

PROPERTY pInitDone : BOOL
GET
pInitDone := bL_InitDone;
END_GET
SET
bL_InitDone := pInitDone;
END_SET
END_PROPERTY

PROPERTY pName : STRING
GET
pName := sL_StateName;
END_GET
SET
sL_StateName := pName;
END_SET
END_PROPERTY

END_FUNCTION_BLOCK

// ---- POUs/Machine/CleaningStation/FB_CleaningProcessStateProduction.TcPOU
FUNCTION_BLOCK FB_CleaningProcessStateProduction EXTENDS FB_CleaningProcessStateBase
VAR_INPUT
END_VAR
VAR_OUTPUT
END_VAR
VAR
END_VAR

METHOD mCleaningOp : BOOL
VAR_INPUT
	sI_Operation : EN_CLEANING_OP;
END_VAR
//Switch to production mode if no operation active
IF I_MachineStatus.pSafetyOk AND I_MachineStatus.pMachineReady AND NOT bL_DevOpActive THEN
  IF sI_Operation = eOPCAPENTER THEN
    I_ParentCallback.mChangeState(EN_Cleaning_State.Capping);
  ELSIF sI_Operation = eOPCAPEXIT THEN
    I_ParentCallback.mChangeState(EN_Cleaning_State.CappingExit);
  ELSIF sI_Operation = eOPCLEAN THEN
    I_ParentCallback.mChangeState(EN_Cleaning_State.Cleaning);
  ELSIF sI_Operation = eOPPURGE THEN
    I_ParentCallback.mChangeState(EN_Cleaning_State.Capping);
  END_IF
END_IF
END_METHOD

METHOD mDevOpDone : BOOL
VAR_INPUT
END_VAR
;//HOA TEST commented: no wait position with pneumatic axis I_ParentCallback.mChangeState(EN_Cleaning_State.Wait);
END_METHOD

METHOD mEntryAction
VAR_INPUT
END_VAR
iL_CurrentStep := 0;

// Launch initial command to bring system to production mode
bL_DevOpActive := I_ParentCallback.mSetMode(EN_CLEANING_OP.eOPGOTOPROD);
END_METHOD

METHOD mProduction : BOOL
VAR_INPUT
END_VAR
//Request production mode - implement in SubClass
mProduction := TRUE;
END_METHOD

METHOD mService : BOOL
VAR_INPUT
END_VAR
//Switch to service mode
IF NOT bL_DevOpActive THEN
	I_ParentCallback.mChangeState(EN_Cleaning_State.Service);
END_IF
END_METHOD

METHOD mStateAction
VAR_INPUT
END_VAR

VAR
	sL_DeviceStatus: ST_CLEANING_DEV_STATUS;
END_VAR
sL_DeviceStatus := I_ParentCallback.pDeviceStatus;

//If not MachineReady go to wait mode
(*HOA TEST commented
IF I_MachineStatus.pSafetyOk AND NOT bL_DevOpActive THEN
	IF NOT I_MachineStatus.pMachineReady THEN
		bL_DevOpActive := I_ParentCallback.mSetMode(EN_CLEANING_OP.eOPGOTOWAIT);
	END_IF
END_IF
*)
IF bL_DevOpActive THEN
	mDevOp();	
END_IF

//If error go to error mode
IF sL_DeviceStatus.bError THEN
	I_ParentCallback.mChangeState(EN_Cleaning_State.Error);
END_IF

SUPER^.pInitDone := TRUE;
END_METHOD

END_FUNCTION_BLOCK

// ---- POUs/Machine/CleaningStation/FB_CleaningProcessStateService.TcPOU
FUNCTION_BLOCK FB_CleaningProcessStateService EXTENDS FB_CleaningProcessStateBase
VAR_INPUT
END_VAR
VAR_OUTPUT
END_VAR
VAR

END_VAR

METHOD mCleaningOp : BOOL
VAR_INPUT
	sI_Operation : EN_CLEANING_OP;
END_VAR
//Switch to production mode if no operation active
IF I_MachineStatus.pSafetyOk AND I_MachineStatus.pMachineReady AND NOT bL_DevOpActive THEN
  IF sI_Operation = eOPCAPENTER THEN
    I_ParentCallback.mChangeState(EN_Cleaning_State.Capping);
  ELSIF sI_Operation = eOPCAPEXIT THEN
    I_ParentCallback.mChangeState(EN_Cleaning_State.CappingExit);
  ELSIF sI_Operation = eOPCLEAN THEN
    I_ParentCallback.mChangeState(EN_Cleaning_State.Cleaning);
  ELSIF sI_Operation = eOPPURGE THEN
    I_ParentCallback.mChangeState(EN_Cleaning_State.Capping);
  END_IF
END_IF
END_METHOD

METHOD mEntryAction
VAR_INPUT
END_VAR
iL_CurrentStep := 0;

// Launch initial command to bring system to service mode
bL_DevOpActive := I_ParentCallback.mSetMode(EN_CLEANING_OP.eOPPREPSERVICE);
END_METHOD

METHOD mProduction : BOOL
VAR_INPUT
END_VAR
//Switch to production mode if no operation active
IF I_MachineStatus.pSafetyOk AND I_MachineStatus.pMachineReady AND NOT bL_DevOpActive THEN
	I_ParentCallback.mChangeState(EN_Cleaning_State.Production);
END_IF
END_METHOD

METHOD mService : BOOL
VAR_INPUT
END_VAR
//Request service mode - implement in SubClass
mService := TRUE;
END_METHOD

METHOD mStateAction
VAR_INPUT
END_VAR

VAR
	sL_DeviceStatus: ST_CLEANING_DEV_STATUS;
END_VAR
sL_DeviceStatus := I_ParentCallback.pDeviceStatus;

IF bL_DevOpActive THEN
	mDevOp();
END_IF

//If error go to error mode
IF sL_DeviceStatus.bError THEN
	I_ParentCallback.mChangeState(EN_Cleaning_State.Error);
END_IF

SUPER^.pInitDone := TRUE;
END_METHOD

END_FUNCTION_BLOCK

// ---- POUs/Machine/CleaningStation/FB_CleaningProcessStateCapping.TcPOU
FUNCTION_BLOCK FB_CleaningProcessStateCapping EXTENDS FB_CleaningProcessStateBase
VAR_INPUT
END_VAR

VAR_OUTPUT
END_VAR

VAR
END_VAR

METHOD mCleaningOp : BOOL
VAR_INPUT
	sI_Operation : EN_CLEANING_OP;
END_VAR
//Set mode and start process when successful
(*HOA TEST
IF NOT bL_DevOpActive THEN
  bL_DevOpActive := I_ParentCallback.mSetMode(sI_Operation);
  mCleaningOp    := TRUE; //report success
END_IF*) mCleaningOp    := TRUE;

//Switch to production mode if no operation active
IF I_MachineStatus.pSafetyOk AND I_MachineStatus.pMachineReady AND NOT bL_DevOpActive THEN
  IF sI_Operation = eOPCAPENTER THEN
    I_ParentCallback.mChangeState(EN_Cleaning_State.Capping);
  ELSIF sI_Operation = eOPCAPEXIT THEN
    I_ParentCallback.mChangeState(EN_Cleaning_State.CappingExit);
  ELSIF sI_Operation = eOPCLEAN THEN
    I_ParentCallback.mChangeState(EN_Cleaning_State.Cleaning);
  ELSIF sI_Operation = eOPPURGE THEN
    I_ParentCallback.mChangeState(EN_Cleaning_State.Capping);
  END_IF
END_IF
END_METHOD

METHOD mEntryAction
VAR_INPUT
END_VAR
iL_CurrentStep := 0;

// Launch initial command to bring system to service mode
bL_DevOpActive := I_ParentCallback.mSetMode(EN_CLEANING_OP.eOPCAPENTER);
END_METHOD

METHOD mProduction : BOOL
VAR_INPUT
END_VAR
//Switch to production mode if no operation active
IF I_MachineStatus.pSafetyOk AND I_MachineStatus.pMachineReady AND NOT bL_DevOpActive THEN
	I_ParentCallback.mChangeState(EN_Cleaning_State.Production);
END_IF
END_METHOD

METHOD mService : BOOL
VAR_INPUT
END_VAR
//Switch to service mode
IF NOT bL_DevOpActive THEN
	I_ParentCallback.mChangeState(EN_Cleaning_State.Service);
END_IF
END_METHOD

METHOD mStateAction
VAR_INPUT
END_VAR

VAR
	sL_DeviceStatus: ST_CLEANING_DEV_STATUS;
END_VAR
sL_DeviceStatus := I_ParentCallback.pDeviceStatus;
SUPER^.pInitDone := TRUE;

IF bL_DevOpActive THEN
	mDevOp();	
END_IF



//If error go to error mode
IF sL_DeviceStatus.bError THEN
	I_ParentCallback.mChangeState(EN_Cleaning_State.Error);
END_IF
END_METHOD

END_FUNCTION_BLOCK

// ---- POUs/Machine/CleaningStation/FB_CleaningProcessStateCappingExit.TcPOU
FUNCTION_BLOCK FB_CleaningProcessStateCappingExit EXTENDS FB_CleaningProcessStateBase
VAR_INPUT
END_VAR

VAR_OUTPUT
END_VAR

VAR
END_VAR

METHOD mCleaningOp : BOOL
VAR_INPUT
	sI_Operation : EN_CLEANING_OP;
END_VAR
//Set mode and start process when successful
(*HOA TEST
IF NOT bL_DevOpActive THEN
  bL_DevOpActive := I_ParentCallback.mSetMode(sI_Operation);
  mCleaningOp    := TRUE; //report success
END_IF*) mCleaningOp    := TRUE;

//Switch to production mode if no operation active
IF I_MachineStatus.pSafetyOk AND I_MachineStatus.pMachineReady AND NOT bL_DevOpActive THEN
  IF sI_Operation = eOPCAPENTER THEN
    I_ParentCallback.mChangeState(EN_Cleaning_State.Capping);
  ELSIF sI_Operation = eOPCAPEXIT THEN
    I_ParentCallback.mChangeState(EN_Cleaning_State.CappingExit);
  ELSIF sI_Operation = eOPCLEAN THEN
    I_ParentCallback.mChangeState(EN_Cleaning_State.Cleaning);
  ELSIF sI_Operation = eOPPURGE THEN
    I_ParentCallback.mChangeState(EN_Cleaning_State.Capping);
  END_IF
END_IF
END_METHOD

METHOD mEntryAction
VAR_INPUT
END_VAR
iL_CurrentStep := 0;

// Launch initial command to bring system to service mode
bL_DevOpActive := I_ParentCallback.mSetMode(EN_CLEANING_OP.eOPCAPEXIT);
END_METHOD

METHOD mProduction : BOOL
VAR_INPUT
END_VAR
//Switch to production mode if no operation active
IF I_MachineStatus.pSafetyOk AND I_MachineStatus.pMachineReady AND NOT bL_DevOpActive THEN
	I_ParentCallback.mChangeState(EN_Cleaning_State.Production);
END_IF
END_METHOD

METHOD mService : BOOL
VAR_INPUT
END_VAR
//Switch to service mode
IF NOT bL_DevOpActive THEN
	I_ParentCallback.mChangeState(EN_Cleaning_State.Service);
END_IF
END_METHOD

METHOD mStateAction
VAR_INPUT
END_VAR

VAR
	sL_DeviceStatus: ST_CLEANING_DEV_STATUS;
END_VAR
sL_DeviceStatus := I_ParentCallback.pDeviceStatus;
SUPER^.pInitDone := TRUE;

IF bL_DevOpActive THEN
	mDevOp();	
END_IF



//If error go to error mode
IF sL_DeviceStatus.bError THEN
	I_ParentCallback.mChangeState(EN_Cleaning_State.Error);
END_IF
END_METHOD

END_FUNCTION_BLOCK

// ---- POUs/Machine/CleaningStation/FB_CleaningProcessStateCleaning.TcPOU
FUNCTION_BLOCK FB_CleaningProcessStateCleaning EXTENDS FB_CleaningProcessStateBase
VAR_INPUT
END_VAR

VAR_OUTPUT
END_VAR

VAR
END_VAR

METHOD mCleaningOp : BOOL
VAR_INPUT
	sI_Operation : EN_CLEANING_OP;
END_VAR
//Set mode and start process when successful
(*HOA TEST
IF NOT bL_DevOpActive THEN
  bL_DevOpActive := I_ParentCallback.mSetMode(sI_Operation);
  mCleaningOp    := TRUE; //report success
END_IF*) mCleaningOp    := TRUE;

//Switch to production mode if no operation active
IF I_MachineStatus.pSafetyOk AND I_MachineStatus.pMachineReady AND NOT bL_DevOpActive THEN
  IF sI_Operation = eOPCAPENTER THEN
    I_ParentCallback.mChangeState(EN_Cleaning_State.Capping);
  ELSIF sI_Operation = eOPCAPEXIT THEN
    I_ParentCallback.mChangeState(EN_Cleaning_State.CappingExit);
  ELSIF sI_Operation = eOPCLEAN THEN
    I_ParentCallback.mChangeState(EN_Cleaning_State.Cleaning);
  ELSIF sI_Operation = eOPPURGE THEN
    I_ParentCallback.mChangeState(EN_Cleaning_State.Capping);
  END_IF
END_IF
END_METHOD

METHOD mEntryAction
VAR_INPUT
END_VAR
iL_CurrentStep := 0;

// Launch initial command to bring system to service mode
bL_DevOpActive := I_ParentCallback.mSetMode(EN_CLEANING_OP.eOPCLEAN);
END_METHOD

METHOD mProduction : BOOL
VAR_INPUT
END_VAR
//Switch to production mode if no operation active
IF I_MachineStatus.pSafetyOk AND I_MachineStatus.pMachineReady AND NOT bL_DevOpActive THEN
	I_ParentCallback.mChangeState(EN_Cleaning_State.Production);
END_IF
END_METHOD

METHOD mService : BOOL
VAR_INPUT
END_VAR
//Switch to service mode
IF NOT bL_DevOpActive THEN
	I_ParentCallback.mChangeState(EN_Cleaning_State.Service);
END_IF
END_METHOD

METHOD mStateAction
VAR_INPUT
END_VAR
IF bL_DevOpActive THEN
	mDevOp();
END_IF

SUPER^.pInitDone := TRUE;
END_METHOD

END_FUNCTION_BLOCK

// ---- POUs/Machine/CleaningStation/FB_CleaningProcessStateError.TcPOU
FUNCTION_BLOCK FB_CleaningProcessStateError EXTENDS FB_CleaningProcessStateBase
VAR_INPUT
END_VAR
VAR_OUTPUT
END_VAR
VAR
END_VAR

METHOD mAbort : BOOL
VAR_INPUT
END_VAR
IF NOT bL_DevOpActive THEN
  bL_DevOpActive := TRUE; //Set to relaunch process
  iL_CurrentStep := 0;
END_IF
I_ParentCallback.mSetMode(EN_Cleaning_OP.eOPEXITERROR);
I_ParentCallback.mDeviceAbort();
END_METHOD

METHOD mAckError : BOOL
VAR_INPUT
END_VAR

VAR
	sL_DeviceStatus: ST_CLEANING_DEV_STATUS;
END_VAR
sL_DeviceStatus := I_ParentCallback.pDeviceStatus;

IF NOT sL_DeviceStatus.bError THEN
  IF NOT SUPER^.pInitDone THEN
    I_ParentCallback.mChangeState(EN_Cleaning_State.Init);
  ELSE  
    I_ParentCallback.mChangeState(EN_Cleaning_State.Service);
  END_IF
END_IF
END_METHOD

METHOD mStateAction
VAR_INPUT
END_VAR

VAR
	sL_DeviceStatus: ST_CLEANING_DEV_STATUS;
END_VAR
sL_DeviceStatus := I_ParentCallback.pDeviceStatus;

SUPER^.pInitDone := sL_DeviceStatus.bRefKnown;

IF bL_DevOpActive THEN
	mDevOp();
END_IF
END_METHOD

END_FUNCTION_BLOCK

// ---- POUs/Machine/CleaningStation/FB_CleaningProcessStateWait.TcPOU
FUNCTION_BLOCK FB_CleaningProcessStateWait EXTENDS FB_CleaningProcessStateBase
VAR_INPUT
END_VAR
VAR_OUTPUT
END_VAR
VAR
END_VAR

METHOD mDevOpDone : BOOL
VAR_INPUT
END_VAR
I_ParentCallback.mChangeState(EN_Cleaning_State.Production);
END_METHOD

METHOD mService : BOOL
VAR_INPUT
END_VAR
//Switch to service mode
IF NOT bL_DevOpActive THEN
	I_ParentCallback.mChangeState(EN_Cleaning_State.Service);
END_IF
END_METHOD

METHOD mStateAction
VAR_INPUT
END_VAR

VAR
	sL_DeviceStatus: ST_CLEANING_DEV_STATUS;
END_VAR
sL_DeviceStatus := I_ParentCallback.pDeviceStatus;

//If MachineReady go to production mode
IF I_MachineStatus.pSafetyOk AND NOT bL_DevOpActive THEN
	IF I_MachineStatus.pMachineReady THEN
		bL_DevOpActive := I_ParentCallback.mSetMode(EN_CLEANING_OP.eOPGOTOPROD);
	END_IF
END_IF

IF bL_DevOpActive THEN
	mDevOp();	
END_IF

//If error go to error mode
IF sL_DeviceStatus.bError THEN
	I_ParentCallback.mChangeState(EN_Cleaning_State.Error);
END_IF
END_METHOD

END_FUNCTION_BLOCK

// ---- POUs/Machine/CleaningStation/FB_CLEANING_PROCESS.TcPOU
FUNCTION_BLOCK FB_CLEANING_PROCESS
(*************************************************************************************************)
(*  FILENAME:    FB_CLEANING_PROCESS.EXP                                                         *)
(*  PROJECT:     CALMAR PUPLC                                                                    *)
(*  COPYRIGHT:   All rights reserved (c) Wifag//Polytype, Fribourg/Switzerland (2016)            *)
(*  ENVIRONMENT: TwinCAT PLC                                                                     *)
(*  VERSION:     <version>                                                                       *)
(*************************************************************************************************)
(*  DESCRIPTION:                                                                   <description> *)
(*     This block controls the cleaning process.                                                 *)
(*     cL_State: cL_IDLE  : (*Idle-State, no operation active*)                                  *)
(*               cL_INIT  : (*Initialize*)                                                       *)
(*               cL_PREP  : (*Prepare*)                                                          *)
(*               cL_START : (*Start*)                                                            *)
(*               cL_STOP  : (*Stop*)                                                             *)
(*     Messaging: - fb_Msg[1] := `eCSy_TestMessageErrorStatus`                                   *)
(*                - fb_Msg[2] := `eCMa_LOCK_CLEANING_MACHINE`                                    *)
(*                                                                                </description> *)
(*************************************************************************************************)

{library public}
VAR_INPUT
(*User commands*)
  bI_UsrPurge                    : BOOL;                         (*User requests purge*)
  bI_UsrStartCapping             : BOOL;                         (*User requests start of capping*)
  bI_UsrStopCapping              : BOOL;                         (*User requests end of capping*)
  bI_UsrClean                    : BOOL;                         (*User requests cleaning*)
  bI_UsrMaintenance              : BOOL;                         (*User requests maintenance*)
  bI_UsrShutter                  : BOOL;                         (*User requests maintenance*)
  bI_UsrAbort                    : BOOL;                         (*User requests abort*)
  bI_UsrAckError                 : BOOL;                         (*User acknowledes error*)
  bI_UsrAutoMode                 : BOOL;                         (*User has selected automatic mode*)
  bI_UsrService                  : BOOL;                         (*User has selected service (1) or print(0) mode*)
  bI_UsrCleanAfterPurge          : BOOL;                         (*Automatically clean after Purge*)
  bI_UsrCleanAfterCapp           : BOOL;                         (*Automatically clean after Capping*)
  bI_UsrPurgeAfterCapp           : BOOL;                         (*Automatically purge after Capping*)
  bI_MachineReady                : BOOL;                         (*Machine ready*)
  bI_CleaningStepEnabled         : ARRAY[1..cL_NB_CLEANSTEPS] OF BOOL;             (*Cleaning step enabled*)
  bI_LockCleaning                : BOOL := FALSE;                (*Lock cleaning*)

(*Device feedback*)
  iI_CfgCleaningPos              : INT;                          (*Number of cleaning positions*)
  sI_CleanDevStatus              : ARRAY[1..cL_NB_CD] OF ST_CLEANING_DEV_STATUS;   (*Initialize operation*)

(*Message system*)
  pC_MsgInterface                : POINTER TO ST_ADS_MSG_IF;     (*Pointer to message interface*)
  iC_BlockId                     : INT;                          (*Message system block ID*)

(*Config*)
  cI_NB_CD                       : INT;                          (*Config number of cleaning devices*)
END_VAR

VAR_OUTPUT
(*Commands*)
  sO_CleanDevCmd                 : ARRAY[1..cL_NB_CD] OF ST_CLEANING_DEV_CMD;      (*Initialize operation*)
  iO_CurrentCleanPos             : INT;                          (*Currently active cleaning position*)

(*Status*)
  bO_CleaningActive              : BOOL;                         (*Any operation active*)
  bO_PurgeActive                 : BOOL;                         (*Purge active*)
  bO_StartCappingActive          : BOOL;                         (*Start of capping active*)
  bO_StopCappingActive           : BOOL;                         (*End of capping active*)
  bO_CleanActive                 : BOOL;                         (*Cleaning active*)
  bO_MaintenanceActive           : BOOL;                         (*Maintenance active*)
  bO_ShutterActive               : BOOL;                         (*Shutter open active*)
  bO_AbortActive                 : BOOL;                         (*Abort active*)
  bO_AckErrorActive              : BOOL;                         (*Acknowledge error active*)

  bO_CmdCleaningCanExec          : BOOL;                         (*Can accept new cleaning commands*)
  bO_CmdCappingCanExec           : BOOL;                         (*Can accept new capping commands*)
  bO_CmdCanExec                  : BOOL;                         (*Can accept new commands other than abort*)
  bO_AbortCanEx                  : BOOL;                         (*Can accept abort command*)
  bO_AckErrorCanEx               : BOOL;                         (*Can accept acknowledge error command*)
END_VAR

{library private}
VAR
  iL_CdCount                     : INT;                          (*Cleaning device counter*)
  cL_State                       : BYTE;                         (*State type*)
  cL_Operation                   : EN_CLEANING_OP;               (*Operation type*)
  bL_ProcessStart                : BOOL;
  iL_CleanStepsDone              : INT;                          (*Cleaning step counter*)
  bL_StepDone                    : BOOL;                         (*The requested step is complete*)
  bL_StateChange                 : BOOL;                         (*The state has changed recently*)
  bL_AllDone                     : BOOL;                         (*All attached axes are done*)
  bL_AllReferenced               : BOOL;                         (*All axes are referenced*)
  bL_AxisError                   : BOOL;                         (*No axis has error*)
  bL_ServiceMode                 : BOOL := TRUE;                 (*Service mode*)
  bL_memServiceMode              : BOOL;                         (*Memory service mode*)
  bL_ServiceModeRequest          : BOOL;                         (*Service mode request*)
  fB_AckErrorHandshake           : FB_FOURCYCLEHANDSHAKE;        (*Acknowledge error*)

  (*Commands*)
  bL_Init                        : BOOL;                         (*Initialize operation*)
  bL_Prep                        : BOOL;                         (*Prepare operation*)
  bL_Start                       : BOOL;                         (*Start operation*)
  bL_Stop                        : BOOL;                         (*Stop operation*)
  bL_Abort                       : BOOL;                         (*Abort operation*)

  (*Message Queue*)
  fB_MsgQueue                    : FB_MSG_QUEUE;                 (*Message queue*)
  fB_MsgHandler                  : FB_MSG_HANDLER;               (*Message handler*)
  sL_MsgConfig                   : ST_MSG_CONFIG;                (*Message config*)
  fB_Msg                         : ARRAY [1..iC_NUM_MSG] OF FB_MESSAGE;  (*Messages*)
END_VAR

VAR CONSTANT
  (*Configuration Placeholders*)
  cL_NB_CD                       : WORD := 5;                    (*Number of cleaning devices*)
  cL_NB_CLEANSTEPS               : WORD := 2;                    (*Number of cleaning steps*)

  (*State*)
  cL_IDLE                        : BYTE := 0;                    (*Idle-State, no operation active*)
  cL_INIT                        : BYTE := 10;                   (*Initialize*)
  cL_PREP                        : BYTE := 20;                   (*Prepare*)
  cL_START                       : BYTE := 30;                   (*Start*)
  cL_STOP                        : BYTE := 40;                   (*Stop*)

  (*Message config*)
  iC_NUM_MSG                     : INT  := 2;                    (*Config number of messages*)
END_VAR

(*Check if devices are done*)
bL_AllDone       := TRUE;
bL_AllReferenced := TRUE;
bL_AxisError     := FALSE;

FOR iL_CdCount := 1 TO cI_NB_CD DO
	IF NOT sI_CleanDevStatus[iL_CdCount].bReady  THEN
		bL_AllDone := FALSE;
	END_IF;

	IF NOT sI_CleanDevStatus[iL_CdCount].bRefKnown  THEN
		bL_AllReferenced := FALSE;
	END_IF;

	IF sI_CleanDevStatus[iL_CdCount].bError THEN
		bL_AxisError := TRUE;
	END_IF;
END_FOR;

IF bL_StateChange THEN
	bL_AllDone := FALSE;
END_IF;

IF NOT bL_AllReferenced THEN
	bL_ServiceModeRequest := TRUE;
	bL_memServiceMode     := FALSE;
ELSE
	bL_ServiceModeRequest := bI_UsrService;
END_IF;

(*StateMachine*)
StateActionLogic();
NextStateLogic();

(*Update Commands*)
iO_CurrentCleanPos := 1 + iL_CleanStepsDone;
FOR iL_CdCount := 1 TO cI_NB_CD DO
	sO_CleanDevCmd[iL_CdCount].bInit      := bL_Init;
	sO_CleanDevCmd[iL_CdCount].bPrep      := bL_Prep;
	sO_CleanDevCmd[iL_CdCount].bStart     := bL_Start;
	sO_CleanDevCmd[iL_CdCount].bStop      := bL_Stop;
	sO_CleanDevCmd[iL_CdCount].bAbort     := bL_Abort;
	sO_CleanDevCmd[iL_CdCount].eOperation := cL_Operation;
	sO_CleanDevCmd[iL_CdCount].bAuto      := bI_UsrAutoMode;
	sO_CleanDevCmd[iL_CdCount].bService   := bL_ServiceMode;
	sO_CleanDevCmd[iL_CdCount].bAckError  := fB_AckErrorHandshake.bO_PlcCmd;
END_FOR;

(*Update Flags*)
IF     cL_State = cL_IDLE
   AND NOT bL_AxisError
   AND bI_UsrAutoMode
   AND bI_UsrService
   AND bL_memServiceMode
THEN
  bO_CmdCanExec           := TRUE;
  IF NOT bI_LockCleaning THEN
    bO_CmdCleaningCanExec := TRUE;
    bO_CmdCappingCanExec  := TRUE;
  ELSE
    bO_CmdCleaningCanExec := FALSE;
    bO_CmdCappingCanExec  := NOT bI_UsrCleanAfterCapp;
  END_IF
ELSE
  bO_CmdCanExec           := FALSE;
  bO_CmdCleaningCanExec   := FALSE;
  bO_CmdCappingCanExec    := FALSE;
END_IF;

IF cL_State <> cL_IDLE AND NOT bL_AxisError THEN
	bO_AbortCanEx := TRUE;
ELSE
	bO_AbortCanEx := FALSE;
END_IF;

bO_AckErrorCanEx               := bL_AxisError;
fB_AckErrorHandshake.bI_AdsCmd := bI_UsrAckError;
fB_AckErrorHandshake.bI_PlcAck := NOT bL_AxisError;

fB_AckErrorHandshake();

bO_AckErrorActive              := fB_AckErrorHandshake.bO_AdsAck;


bO_PurgeActive        := FALSE;
bO_StartCappingActive := FALSE;
bO_StopCappingActive  := FALSE;
bO_CleanActive        := FALSE;
bO_MaintenanceActive  := FALSE;
bO_ShutterActive      := FALSE;

CASE cL_Operation OF
	eOPPURGE:         bO_PurgeActive        := TRUE;
	eOPCAPENTER:      bO_StartCappingActive := TRUE;
	eOPCAPEXIT:       bO_StopCappingActive  := TRUE;
	eOPCLEAN:         bO_CleanActive        := TRUE;
	eOPMAINT:         bO_MaintenanceActive  := TRUE;
	eOPSHUTTEROPEN:   bO_ShutterActive      := TRUE;
END_CASE;

bO_AbortActive := bL_Abort;

(*Message Queue --------------------------------------------------------------------*)
fB_MsgHandler();

(*eCSy_TestMessageErrorStatus
IF ERROR THEN
  fB_Msg[1].bI_Status := TRUE;
ELSE
  fB_Msg[1].bI_Status := FALSE;
END_IF;
fB_Msg[1]();
*)
fB_Msg[2](bI_Status := bI_LockCleaning);

fB_MsgQueue();

(********************************* END OF FB *****************************************************)

ACTION Init:
(*Messages*)
sL_MsgConfig.bI_Enable       := TRUE;
sL_MsgConfig.pI_FbMsgHandler := ADR(fB_MsgHandler);
fB_MsgHandler.pI_MsgQueue    := ADR(fB_MsgQueue);
fB_MsgQueue.pI_MsgInterface  := pC_MsgInterface;
fB_MsgQueue.cI_MaxElement    := 5;

fB_Msg[1].iI_MsgLocation     := iC_BlockId;
fB_Msg[1].pI_MsgConfig       := ADR(sL_MsgConfig);
fB_Msg[1].iI_MsgNumber       := eCSy_TestMessageErrorStatus;

fB_Msg[2].iI_MsgLocation     := iC_BlockId;
fB_Msg[2].pI_MsgConfig       := ADR(sL_MsgConfig);
fB_Msg[2].iI_MsgNumber       := eCMa_LOCK_CLEANING_MACHINE;

(********************************* END OF ACTION *************************************************)
END_ACTION

ACTION NextStateLogic:
(*Next state logic -----------------------------------------------------------------*)

CASE cL_State OF
	cL_IDLE: 		(*No active operation*)
		IF bL_ProcessStart AND bI_MachineReady AND NOT bL_AxisError THEN		(*Start process*)
			cL_State       := cL_INIT;
			bL_StateChange := TRUE;

			(*Select Operation*)
			IF bI_UsrPurge THEN
				cL_Operation := eOPPURGE;
			ELSIF bI_UsrClean THEN
				iL_CleanStepsDone := 0;
				WHILE bI_CleaningStepEnabled[iL_CleanStepsDone + 1] = FALSE AND (iL_CleanStepsDone < iI_CfgCleaningPos) DO
					iL_CleanStepsDone := iL_CleanStepsDone + 1;
				END_WHILE;

				IF (iL_CleanStepsDone >= iI_CfgCleaningPos) OR bI_CleaningStepEnabled[iL_CleanStepsDone + 1] = FALSE THEN
					cL_Operation := eNOP;
				ELSE
					cL_Operation := eOPCLEAN;
				END_IF;

			ELSIF bI_UsrStartCapping THEN
				cL_Operation := eOPCAPENTER;
			ELSIF bI_UsrStopCapping THEN
				cL_Operation := eOPCAPEXIT;
			ELSIF bI_UsrMaintenance THEN
				cL_Operation := eOPMAINT;
			ELSIF bI_UsrShutter THEN
				cL_Operation := eOPSHUTTEROPEN;
			ELSE
				cL_Operation := eNOP;
			END_IF;
		ELSIF bL_ServiceModeRequest AND NOT bL_memServiceMode AND bI_MachineReady AND NOT bL_AxisError THEN	(*Enter Service*)
			IF NOT bL_AllReferenced THEN
				cL_Operation := eOPSTARTUP;
			ELSE
				cL_Operation := eOPPREPSERVICE;
			END_IF;

			cL_State       := cL_INIT;
			bL_StateChange := TRUE;
		ELSIF NOT bL_ServiceModeRequest AND bL_memServiceMode AND bI_MachineReady	AND NOT bL_AxisError THEN(*Enter Print*)
			cL_Operation   := eOPENDSERVICE;
			cL_State       := cL_INIT;
			bL_StateChange := TRUE;
		ELSE
			cL_State       := cL_IDLE;
			bL_StateChange := FALSE;
			cL_Operation   := eNOP;
		END_IF;

	cL_INIT: 		(*Initialize system*)
		IF bL_StepDone THEN 	(**)
			cL_State       := cL_PREP;
			bL_StateChange := TRUE;
		ELSE										(**)
			cL_State       := cL_INIT;
			bL_StateChange := FALSE;
		END_IF;

	cL_PREP: 		(*Prepare system*)
		IF bL_StepDone THEN 	(**)
			cL_State       := cL_START;
			bL_StateChange := TRUE;
		ELSE										(**)
			cL_State       := cL_PREP;
			bL_StateChange := FALSE;
		END_IF;

	cL_START: (*Start process*)
		IF bL_StepDone THEN
			cL_State       := cL_STOP;
			bL_StateChange := TRUE;
		ELSE
			cL_State       := cL_START;
			bL_StateChange := FALSE;
		END_IF;

	cL_STOP: (*Stop process*)
		IF bL_StepDone THEN
			IF cL_Operation = eOPCLEAN THEN
					iL_CleanStepsDone := iL_CleanStepsDone + 1;
				WHILE bI_CleaningStepEnabled[iL_CleanStepsDone + 1] = FALSE AND (iL_CleanStepsDone < iI_CfgCleaningPos) DO
					iL_CleanStepsDone := iL_CleanStepsDone + 1;
				END_WHILE;

				IF iL_CleanStepsDone >= iI_CfgCleaningPos THEN
					cL_State          := cL_IDLE;
					iL_CleanStepsDone := 0;
				ELSE
					cL_State          := cL_INIT;
				END_IF;

				bL_StateChange      := TRUE;
			ELSIF cL_Operation = eOPPURGE AND bI_UsrCleanAfterPurge THEN
					iL_CleanStepsDone := 0;
					WHILE bI_CleaningStepEnabled[iL_CleanStepsDone + 1] = FALSE AND (iL_CleanStepsDone < iI_CfgCleaningPos) DO
						iL_CleanStepsDone := iL_CleanStepsDone + 1;
					END_WHILE;

					IF (iL_CleanStepsDone >= iI_CfgCleaningPos) OR bI_CleaningStepEnabled[iL_CleanStepsDone + 1] = FALSE THEN
						cL_State     := cL_IDLE;
					ELSE
						cL_Operation := eOPCLEAN;
						cL_State     := cL_INIT;
					END_IF;

					bL_StateChange := TRUE;
			ELSIF cL_Operation = eOPCAPEXIT AND bI_UsrCleanAfterCapp THEN
					IF (iL_CleanStepsDone >= iI_CfgCleaningPos) OR bI_CleaningStepEnabled[iL_CleanStepsDone + 1] = FALSE THEN
						cL_State     := cL_IDLE;
					ELSE
						cL_Operation := eOPCLEAN;
						cL_State     := cL_INIT;
					END_IF;

					bL_StateChange := TRUE;
			ELSIF cL_Operation = eOPCAPEXIT AND bI_UsrPurgeAfterCapp THEN
					cL_State       := cL_INIT;
					bL_StateChange := TRUE;
					cL_Operation   := eOPPURGE;
			ELSE
				cL_State       := cL_IDLE;
				bL_StateChange := TRUE;
			END_IF;
		ELSE
			cL_State       := cL_STOP;
			bL_StateChange := FALSE;
		END_IF;
END_CASE;

IF bI_UsrAbort OR bL_AxisError THEN
	cL_State          := cL_IDLE;
	cL_Operation      := eNOP;
	bL_StateChange    := TRUE;
	iL_CleanStepsDone := 0;
END_IF;

(********************************* END OF ACTION *************************************************)
END_ACTION

ACTION StateActionLogic:
(*State action logic -----------------------------------------------------------------*)

CASE cL_State OF
	cL_IDLE: 		(*No active operation*)
		IF bI_UsrPurge THEN
			bL_ProcessStart	:= TRUE;
		ELSIF bI_UsrClean THEN
			bL_ProcessStart	:= TRUE;
		ELSIF bI_UsrStartCapping OR bI_UsrStopCapping THEN
			bL_ProcessStart	:= TRUE;
		ELSIF bI_UsrMaintenance THEN
			bL_ProcessStart	:= TRUE;
		ELSIF bI_UsrShutter THEN
			bL_ProcessStart	:= TRUE;
		ELSE
			bL_ProcessStart	:= FALSE;
		END_IF;
		bL_StepDone       := FALSE;
		bO_CleaningActive := FALSE;

	cL_INIT: 		(*Initialize system*)
		IF bL_StateChange THEN
			bL_StepDone  := FALSE;
			bL_Init			 := TRUE;

			IF cL_Operation = eOPPREPSERVICE OR cL_Operation = eOPSTARTUP THEN
				bL_ServiceMode := TRUE;
			END_IF;

		ELSE
			bL_StepDone  := bL_AllDone AND NOT bL_Init;	(*Delay by one cycle*)
			bL_Init			 := FALSE;
		END_IF;
		bO_CleaningActive := TRUE;

	cL_PREP: 		(*Prepare system*)
		IF bL_StateChange THEN
			bL_StepDone  := FALSE;
			bL_Prep			 := TRUE;
		ELSE
			bL_StepDone  := bL_AllDone AND NOT bL_Prep;	(*Delay by one cycle*)
			bL_Prep		 	 := FALSE;
		END_IF;
		bO_CleaningActive := TRUE;

	cL_START: (*Start process*)
		IF bL_StateChange THEN
			bL_StepDone  := FALSE;
			bL_Start		 := TRUE;
		ELSE
			bL_StepDone  := bL_AllDone AND NOT bL_Start;	(*Delay by one cycle*)
			bL_Start	 	 := FALSE;
		END_IF;
		bO_CleaningActive := TRUE;

	cL_STOP: (*Stop process*)
		IF bL_StateChange THEN
			bL_StepDone  := FALSE;
			bL_Stop			 := TRUE;

			IF cL_Operation = eOPENDSERVICE THEN
				bL_ServiceMode    := FALSE;
				bL_memServiceMode := FALSE;
			END_IF;

			IF cL_Operation = eOPPREPSERVICE OR cL_Operation = eOPSTARTUP THEN
				bL_memServiceMode := TRUE;
			END_IF;

		ELSE
			bL_StepDone  := bL_AllDone AND NOT bL_Stop;	(*Delay by one cycle*)
			bL_Stop		 	 := FALSE;
		END_IF;
		bO_CleaningActive := TRUE;
END_CASE;

IF bI_UsrAbort OR bL_Abort THEN
	bL_Init  := FALSE;
	bL_Prep  := FALSE;
	bL_Start := FALSE;
	bL_Stop  := FALSE;
	IF bL_AllDone THEN
		bL_StepDone := TRUE;
		bL_Abort    := FALSE;
	ELSE
		bL_StepDone := TRUE;
		bL_Abort    := TRUE;
	END_IF;
ELSE
	bL_Abort      := FALSE;
END_IF;

IF bL_AxisError THEN
	bL_Init  := FALSE;
	bL_Prep  := FALSE;
	bL_Start := FALSE;
	bL_Stop  := FALSE;
END_IF;

(********************************* END OF ACTION *************************************************)
END_ACTION

END_FUNCTION_BLOCK

// ---- POUs/Machine/CleaningStation/FB_Cleaning_ValvePump.TcPOU
FUNCTION_BLOCK FB_Cleaning_ValvePump EXTENDS FB_CleanDevice
VAR_INPUT
END_VAR

VAR_OUTPUT
  bO_VacuumValve                  AT %Q* : BOOL;     (*Enable vacuum valve for CleaningStation*)

  bO_VacuumPump                   AT %Q* : BOOL;     (*Enable vacuum pump for CleaningStation*)
  wO_SetPointVacuumPump           AT %Q* : WORD;     (*Vacuum pump set point*)

  bO_CleanerPump                  AT %Q* : BOOL;     (*Enable cleaner pump for CleaningStation*)
  wO_SetPointCleanerPump          AT %Q* : WORD;     (*Cleaner pump set point*)
END_VAR

VAR
  _bManuEmptyTub                         : BOOL;     (*Manually empty tub*)

  bL_VacuumValve                         : BOOL;     (*Enable vacuum valve for CleaningStation*)

  bL_VacuumPump                          : BOOL;     (*Enable vacuum pump for CleaningStation*)
  lL_SetPointVacuumPump                  : DINT;     (*Vacuum pump set point [%]*)

  bL_CleanerPump                         : BOOL;     (*Enable cleaner pump for CleaningStation*)
  lL_SetPointCleanerPump                 : DINT;     (*Cleaner pump set point [%]*)

  fb_TonCleanerPumpOffset                : TON;
  fb_TonVacuumPumpDelay                  : TON;
END_VAR

VAR PERSISTENT
  lR_AnalogMaxDigitVacuumPump            : DINT := 16383;  (*Max value analog-output in digit (32767 = 10V)*)
  lR_SetPoint1VacuumPump                 : DINT;     (*Vacuum pump set point #1 [%]*)
  lR_SetPoint2VacuumPump                 : DINT;     (*Vacuum pump set point #2 [%]*)
  lR_SetPoint3VacuumPump                 : DINT;     (*Vacuum pump set point #3 [%]*)
  lR_SetPoint4VacuumPump                 : DINT;     (*Vacuum pump set point #4 [%]*)
  lR_AnalogMaxDigitCleanerPump           : DINT := 16383;  (*Max value analog-output in digit (32767 = 10V)*)
  lR_SetPoint1CleanerPump                : DINT;     (*Cleaner pump set point #1 [%]*)
  lR_SetPoint2CleanerPump                : DINT;     (*Cleaner pump set point #2 [%]*)
  lR_SetPoint3CleanerPump                : DINT;     (*Cleaner pump set point #3 [%]*)
  lR_SetPoint4CleanerPump                : DINT;     (*Cleaner pump set point #4 [%]*)

  tR_CleanerPumpOffset                   : TIME := T#4S;
  tR_VacuumPumpDelay                     : TIME := T#1S;
  tR_VacuumPumpEmptyBin                  : TIME := T#15S;
END_VAR

METHOD mCleaning : BOOL
VAR_INPUT
  iI_Step : INT;
END_VAR
//Abort: Stop pumps and return
IF bL_AbortReq THEN
  bL_Busy        := FALSE;
  bL_Ready       := TRUE;
  bL_VacuumValve := FALSE;
  bL_VacuumPump  := FALSE;
  bL_CleanerPump := FALSE;
  mSetOutput();
  RETURN;
END_IF

//Normal operation
CASE iI_Step OF
  0: //Init - Check if axis is not activated, restore safety
    fb_TonCleanerPumpOffset(IN := FALSE, PT := tR_CleanerPumpOffset);
    fb_TonVacuumPumpDelay  (IN := FALSE, PT := tR_VacuumPumpDelay);

    bL_Busy := FALSE;

  1: //Wait for PU axis to lift
    bL_Busy := FALSE;
    
  2: //Wait for CU axis to move out
    bL_Busy := FALSE;
    
  3: //Wait for PU axis to lower
    bL_Busy := FALSE;
    
  4: //Ensure CH axis is at starting position
    bL_Busy := FALSE;

  5: //Move CH to clean start position
    bL_Busy := FALSE;

  6: //Wait until cleaning equipment ready
    bL_VacuumValve         := TRUE;

    bL_VacuumPump          := TRUE;
    lL_SetPointVacuumPump  := lR_SetPoint1VacuumPump;

    bL_CleanerPump         := TRUE;
    lL_SetPointCleanerPump := lR_SetPoint1CleanerPump;
    
    mSetOutput();

    (*Delay cleaner pump for a good start-up.*)
    fb_TonCleanerPumpOffset(IN := TRUE, PT := tR_CleanerPumpOffset);
    bL_Busy := NOT fb_TonCleanerPumpOffset.Q;
    
  7: //Cleaning
    bL_Busy := FALSE;
    
  8: //Wait until cleaning equipment ready
    bL_VacuumValve         := TRUE;

    bL_VacuumPump          := TRUE;
    lL_SetPointVacuumPump  := lR_SetPoint1VacuumPump;

    bL_CleanerPump         := FALSE;
    lL_SetPointCleanerPump := lR_SetPoint1CleanerPump;
    
    mSetOutput();

    bL_Busy := FALSE;
    
  9: //Move CH to end position
    (*Off delay vacuum pump.*)
    fb_TonVacuumPumpDelay(IN := TRUE, PT := tR_VacuumPumpDelay);
    bL_Busy := NOT fb_TonVacuumPumpDelay.Q;
    
  10: //Wait for PU axis to lift
    bL_VacuumValve := FALSE;
    bL_VacuumPump  := FALSE;
    mSetOutput();

    bL_Busy := FALSE;
    
  11: //Move CH back to start 
    bL_VacuumValve         := FALSE;

    bL_VacuumPump          := TRUE;
    lL_SetPointVacuumPump  := lR_SetPoint1VacuumPump;

    bL_CleanerPump         := FALSE;
    lL_SetPointCleanerPump := lR_SetPoint1CleanerPump;
    
    mSetOutput();

    bL_Busy := FALSE;
    
  12: //End
    bL_VacuumValve := FALSE;
    bL_VacuumPump  := FALSE;
    mSetOutput();

    bL_Busy := FALSE;
  
  ELSE
    bL_Busy := FALSE;    
END_CASE
END_METHOD

METHOD mManuSetCleanerPump
VAR_INPUT
  bI_CleanerPump                         : BOOL;     (*Enable cleaner pump for CleaningStation*)
  bI_VacuumPump                          : BOOL;     (*Enable vacuum pump for CleaningStation*)
  wI_SetPointCleanerPump                 : DINT;     (*Cleaner pump set point*)
END_VAR
IF bI_CleanerPump THEN
  bO_CleanerPump         := TRUE;
  wO_SetPointCleanerPump := DINT_TO_WORD(lR_AnalogMaxDigitCleanerPump * wI_SetPointCleanerPump / 100);

  bO_VacuumPump          := bI_VacuumPump;                                                              
  wO_SetPointVacuumPump  := DINT_TO_WORD(lR_AnalogMaxDigitVacuumPump);
ELSE
  bO_CleanerPump         := FALSE;
  bO_VacuumPump          := FALSE;
END_IF
END_METHOD

METHOD mProduction : BOOL
VAR_INPUT
  iI_Step : INT;
END_VAR
//Abort: Stop whereever axis is and return
IF bL_AbortReq THEN
  bL_Busy        := FALSE;
  bL_Ready       := TRUE;
  bL_VacuumValve := FALSE;
  bL_VacuumPump  := FALSE;
  bL_CleanerPump := FALSE;
  mSetOutput();
  RETURN;
END_IF

//Normal operation
CASE iI_Step OF
  0: //Init - Check if axis is not activated, restore safety
    fb_TonCleanerPumpOffset(IN := FALSE, PT := tR_VacuumPumpEmptyBin);

    bL_Busy := FALSE;

  1: //Wait for PU axis to lift
    bL_Busy := FALSE;
    
  2: //Wait for CU axis to move out & empty bin
    (*Timer vacuum pump to empty bin.*)
    fb_TonCleanerPumpOffset(IN := TRUE, PT := tR_VacuumPumpEmptyBin);

    bL_VacuumValve         := FALSE;

    bL_VacuumPump          := NOT fb_TonCleanerPumpOffset.Q;
    lL_SetPointVacuumPump  := lR_SetPoint1VacuumPump;

    mSetOutput();

    bL_Busy := FALSE;
    
  3: //Wait for PU axis to lower
    (*Timer vacuum pump to empty bin.*)
    fb_TonCleanerPumpOffset(IN := TRUE, PT := tR_VacuumPumpEmptyBin);

    bL_VacuumValve := FALSE;
    bL_VacuumPump  := NOT fb_TonCleanerPumpOffset.Q;
    mSetOutput();

    bL_Busy := NOT fb_TonCleanerPumpOffset.Q;
    
  4: //End
    bL_VacuumValve := FALSE;
    bL_VacuumPump  := FALSE;
    mSetOutput();

    bL_Busy := FALSE;

  ELSE
    bL_Busy := FALSE;    
END_CASE
END_METHOD

METHOD mSetOutput
VAR_INPUT
END_VAR
bO_VacuumValve         := bL_VacuumValve;

bO_VacuumPump          := bL_VacuumPump;
wO_SetPointVacuumPump  := DINT_TO_WORD(lR_AnalogMaxDigitVacuumPump * lL_SetPointVacuumPump / 100);

bO_CleanerPump         := bL_CleanerPump;
wO_SetPointCleanerPump := DINT_TO_WORD(lR_AnalogMaxDigitCleanerPump * lL_SetPointCleanerPump / 100);
END_METHOD

PROPERTY pManuEmptyTub : BOOL
GET
pManuEmptyTub := _bManuEmptyTub;
END_GET
SET
_bManuEmptyTub := pManuEmptyTub;
IF _bManuEmptyTub THEN
  bO_VacuumValve         := FALSE;
  bO_VacuumPump          := TRUE;
  wO_SetPointVacuumPump  := DINT_TO_WORD(lR_AnalogMaxDigitVacuumPump);
ELSE
  bO_VacuumValve         := FALSE;
  bO_VacuumPump          := FALSE;
END_IF
END_SET
END_PROPERTY

END_FUNCTION_BLOCK

// ---- POUs/Machine/CleaningStation/FB_CU_MOTION_CTRL.TcPOU
FUNCTION_BLOCK FB_CU_MOTION_CTRL
(******************************************************************************************)
(*  FILENAME:     FB_CU_MOTION_CTRL                                                       *)
(*  PROJECT:      Steinemann                                                              *)
(*  COPYRIGHT:    Wifag-Polytype                                                          *)
(*  ENVIRONMENT:  TwinCat2, v2.11                                                         *)
(*  VERSION:      1.0                                                                     *)
(*  DESCRIPTION:                                                                          *)
(*    This Function is to control the mouvements of the Printer Unit                      *)
(*    on the X Axis. It will control the operation type and the service                   *)
(*    mode to send motion commands to the axis                                            *)
(*  AUTHOR:      M: BOYRAZ, GoConcept                                                     *)
(******************************************************************************************)
(*  MODIFICATIONS:                                                                        *)
(******************************************************************************************)
(*  Date        Authtor   Descriptons                                                     *)
(*  01.05.2014  FAF       Major redesign                                                  *)
(******************************************************************************************)

VAR_INPUT
(*Commands from Cleaning Process Controller*)
	sI_CleanDevCmd                  : ST_CLEANING_DEV_CMD;	(*Initialize operation*)
	iI_CurrentCleanPos              :	INT := 0;	(*Currently active cleaning position*)

(*Settings*)
	sI_SpeedDef_X                   : ST_SPEEDS;
	fI_CurrentPosition              : REAL;					(*Current axis position*)
	fI_ParkPosition                 : REAL := 0.0;		(*Park Positon (Production Mode)*)
	fI_CappPurgPosition             : REAL := 0.0;		(*Capping/Purge (Service Mode)*)
	fI_CleanRowPositions            : ARRAY[1..cL_NB_CLEANPOS] OF REAL;
	fI_PositionTolerance            : REAL := 0.0001;(*Service position (Service Mode)*)
  fI_SetPositionValue             : REAL := 0.0;    (*Set position value [m]*)

(*User Commands*)
	sI_ManualCommands               : ST_MANUAL_CMD;
	bI_AckFault                     : BOOL;	(* Acknowledge errors*)
	bI_Enable                       : BOOL;	(* Enable PrintUnit axis*)

(*Machine Flags*)
	bI_DeviceOnline                 : BOOL;	(*Check link to device*)
	bI_ReferenceSensor              : BOOL;	(*Reference Sensor activated*)
	bI_SystemReady                  : BOOL;	(*General ready flag*)
	bI_MachineReady                 : BOOL;	(*Machine ready = go to print if not in service*)
	bI_MovementAllowed              : BOOL;	(*No collision danger*)
	bI_HomingAllowed                : BOOL;	(*Homing allowed*)
	bI_SafetyOk                     : BOOL;	(*Safety ok for movement*)
	eI_ELmodule_State               : EN_EL7201_STATE;	(*Feedback from Axis*)
	bI_MoveOk                       : BOOL;

	pC_MsgInterface                 : POINTER TO ST_ADS_MSG_IF;
	iC_BlockId                      : INT;
END_VAR

VAR_OUTPUT
	sO_ClnUnit_Mvt_Status           : ST_CU_STATUS;
	sO_CleanDevStatus               : ST_CLEANING_DEV_STATUS;	(*Initialize operation*)

	fO_TargetPosition               : REAL;	(*Target position for axis*)
	fO_SpeedLimit                   : REAL;	(*Speed limit for axis*)
	bO_MoveEnable                   : BOOL;	(*Move enable for axis*)
	bO_RegActive                    : BOOL;	(*Close control loop for axis*)
	bO_FaultReset                   : BOOL;	(*Fault reset for axis*)
	bO_SetPosition                  : BOOL; (*Reset Encoder*)
	bO_PositionUnknown              : BOOL; (*Position of axis is unknown*)
END_VAR

VAR
	bL_SafeRunningCondition         : BOOL;
	bL_SafeMoveNeg                  : BOOL;
	bL_SafeMovePos                  : BOOL;

	bL_AxisReady                    : BOOL;	(*Axis has no pending operation*)
	bL_PrintReady                   : BOOL;	(*Axis is ready to print*)
	bL_AfterHoming                  : BOOL;	(*Flag is set when RefUnknown*)

	wL_ErrorCode                    : WORD;

	bL_InPosition_For_Cleaning      : BOOL;
	bL_InPosition_For_CappPurg      : BOOL;
	bL_InPosition_For_Parking       : BOOL;

	bL_MotionActive                 : BOOL;
	tL_TimerSurv                    : TON;			(* Timer for Motorization check *)

	bL_Ref_Known                    : BOOL := FALSE;
	bL_MoveStarted                  : BOOL := FALSE;
	bL_MoveStartRequested           : BOOL := FALSE;
	bL_MoveDone                     : BOOL := FALSE;

	(*Memory registers*)
	bL_mem_MotionActive             : BOOL;
	bL_memRefSensor                 : BOOL;
	bL_memAckFault                  : BOOL;
	fL_memX_Position                : REAL;
	bL_mem_MoveEnable               : BOOL;
	bL_FirstRun                     : BOOL := TRUE;

	(*Messaging*)
 	fB_MsgQueue                     : FB_MSG_QUEUE;
	fB_MsgHandler                   : FB_MSG_HANDLER;
	sL_MsgConfig                    : ST_MSG_CONFIG;
	fB_Msg                          : ARRAY [1..iC_NUM_MSG] OF FB_MESSAGE;
END_VAR

VAR CONSTANT
	cL_NB_CLEANPOS                  : WORD := 2;						(*Number of cleaning positions*)
	iC_NUM_MSG                      : INT  := 1;
END_VAR

tL_TimerSurv.PT := T#3s;
tL_TimerSurv();

(*----------------------------------------------------------------------------------------------------------------------------------------------- *)
(*Position detection*)
(*----------------------------------------------------------------------------------------------------------------------------------------------- *)

IF     fI_CurrentPosition >= (fI_CappPurgPosition - fI_PositionTolerance)
   AND fI_CurrentPosition <= (fI_CappPurgPosition + fI_PositionTolerance)
THEN
  bL_InPosition_For_CappPurg := TRUE;
  bL_InPosition_For_Parking  := FALSE;
  bL_InPosition_For_Cleaning := FALSE;
ELSIF  fI_CurrentPosition >= (fI_ParkPosition - fI_PositionTolerance)
   AND fI_CurrentPosition <= (fI_ParkPosition + fI_PositionTolerance)
THEN
  bL_InPosition_For_CappPurg := FALSE;
  bL_InPosition_For_Parking  := TRUE;
  bL_InPosition_For_Cleaning := FALSE;
ELSE
  bL_InPosition_For_CappPurg := FALSE;
  bL_InPosition_For_Parking  := FALSE;

  IF     fI_CurrentPosition >= (fI_CleanRowPositions[iI_CurrentCleanPos] - fI_PositionTolerance)
     AND fI_CurrentPosition <= (fI_CleanRowPositions[iI_CurrentCleanPos] + fI_PositionTolerance)
  THEN
    bL_InPosition_For_Cleaning := TRUE;
  ELSE
    bL_InPosition_For_Cleaning := FALSE;
  END_IF;
END_IF;

(*----------------------------------------------------------------------------------------------------------------------------------------------- *)
(*----------------------------------- Safe Running Conditions  For Printing Unit  --------------------------------------------------------------- *)
(*----------------------------------------------------------------------------------------------------------------------------------------------- *)
IF bI_Enable AND bI_SystemReady AND bI_DeviceOnline AND bI_SafetyOk AND (wL_ErrorCode = 0 OR wL_ErrorCode.5 OR wL_ErrorCode.6)THEN	(*Dont check limit switch here*)
	bL_SafeRunningCondition := TRUE;
ELSE
	bL_SafeRunningCondition := FALSE;
END_IF;
bL_SafeMoveNeg := bL_SafeRunningCondition AND NOT bI_ReferenceSensor AND bI_MovementAllowed;
bL_SafeMovePos := bL_SafeRunningCondition AND bI_MovementAllowed;

IF NOT bI_DeviceOnline THEN
	bL_Ref_Known := FALSE;				(*Reset Reference when link to device is lost, e.g. when machine power off*)
END_IF;

(*----------------------------------------------------------------------------------------------------------------------------------------------- *)
(*------------------------------------------- Motion Control For the Cleaning Unit   ------------------------------------------------------------ *)
(*----------------------------------------------------------------------------------------------------------------------------------------------- *)
IF NOT bL_Ref_Known THEN	(* if the X axis hasn't been initialized with Ref Sensor*)
	bL_AxisReady   := FALSE;
	bL_AfterHoming := TRUE;
	IF bI_ReferenceSensor AND NOT bL_memRefSensor AND NOT bL_Ref_Known THEN		(**)
		bL_Ref_Known    := TRUE;											(* When the sensor is activated, Save the correction value*)
		bL_MotionActive := FALSE;										(**)
		bO_SetPosition  := TRUE;											(*Initialize Position to Preset Value*)
		bL_AxisReady    := TRUE;

		fO_TargetPosition := fI_SetPositionValue;
	ELSE
		IF bI_ReferenceSensor AND bL_memRefSensor THEN
			fO_TargetPosition := fI_CurrentPosition + 0.01;			(*@@@@CONST, change to JOG_NEGATIVE*);					(* *)
			fO_SpeedLimit     := sI_SpeedDef_X.fP_ServiceSpeed;	(* Start backward motion, the motor will run until Ref Sensor is ON*)
			bL_MotionActive   := bI_HomingAllowed;								(* *)
			bO_SetPosition    := FALSE;
		ELSE
			fO_TargetPosition := -100.0											(*@@@@CONST, change to JOG_NEGATIVE*);					(* *)
			fO_SpeedLimit     := sI_SpeedDef_X.fP_ServiceSpeed;	(* Start backward motion, the motor will run until Ref Sensor is ON*)
			bL_MotionActive   := bI_HomingAllowed;								(* *)
			bO_SetPosition    := FALSE;
		END_IF;
	END_IF;																(**)
ELSE	(* If the X axis has been initialized *)
	IF sI_CleanDevCmd.bService THEN
		ServiceMode();
	ELSE
		ProductionMode();
	END_IF;
END_IF;
bL_memRefSensor := bI_ReferenceSensor;				(* Memorization of the Ref Sensor state ffor edge detection*)



(*----------------------------------------------------------------------------------------------------------------------- *)
(*----------------------------------- Output Structure Data Update  ----------------------------------------------------- *)
(*----------------------------------------------------------------------------------------------------------------------- *)
sO_CleanDevStatus.bBusy     := NOT(bL_AxisReady);
sO_CleanDevStatus.bReady    := bL_AxisReady;
sO_CleanDevStatus.bRefKnown := NOT bO_PositionUnknown;

IF wL_ErrorCode = 0 THEN
	sO_CleanDevStatus.bError := FALSE;
ELSE
	sO_CleanDevStatus.bError := TRUE;
END_IF;

sO_ClnUnit_Mvt_Status.bO_Active              := bI_Enable;
sO_ClnUnit_Mvt_Status.bO_Busy                := bO_MoveEnable;
sO_ClnUnit_Mvt_Status.bO_Ready               := bL_AxisReady;
sO_ClnUnit_Mvt_Status.fO_Position            := fI_CurrentPosition;
sO_ClnUnit_Mvt_Status.bO_InPosition_Capping  := bL_InPosition_For_CappPurg;
sO_ClnUnit_Mvt_Status.bO_InPosition_Cleaning := bL_InPosition_For_Cleaning;
sO_ClnUnit_Mvt_Status.bO_InPosition_Parking  := bL_InPosition_For_Parking;
sO_ClnUnit_Mvt_Status.bO_InPosition_Purging  := bL_InPosition_For_CappPurg;
sO_ClnUnit_Mvt_Status.bO_ReferenceKnown      := bL_Ref_Known;
sO_ClnUnit_Mvt_Status.wO_FaultCode           := wL_ErrorCode;

bO_FaultReset                                := bI_AckFault (*OR fb_MsgQueue.bO_ReceiptMessage*) OR sI_CleanDevCmd.bAckError;

IF wL_ErrorCode = 0 THEN
	sO_ClnUnit_Mvt_Status.bO_Error := FALSE;
ELSE
	sO_ClnUnit_Mvt_Status.bO_Error := TRUE;
END_IF;

bO_RegActive := bI_Enable AND bL_SafeRunningCondition;

IF fI_CurrentPosition < fO_TargetPosition THEN			(*  is UP Mouvement *)
	bO_MoveEnable := bL_MotionActive AND bL_SafeMovePos;
ELSE											(*  is DOWN Mouvement *)
	bO_MoveEnable := bL_MotionActive AND bL_SafeMoveNeg;
END_IF;

IF bL_MotionActive AND NOT bL_mem_MotionActive THEN
	bL_MoveStartRequested := TRUE;
	bL_MoveStarted        := FALSE;
	bL_MoveDone           := FALSE;
END_IF;

IF bO_MoveEnable AND NOT bL_mem_MoveEnable AND bL_MoveStartRequested THEN
	bL_MoveStarted := TRUE;
	bL_MoveDone    := FALSE;
ELSIF bL_MoveStarted THEN
	IF bI_MoveOk OR sI_CleanDevCmd.bAbort THEN
		bL_MoveDone           := TRUE;
		bL_MoveStarted        := FALSE;
		bL_MoveStartRequested := FALSE;
	END_IF;
END_IF;

(*----------------------------------------------------------------------------------------------------------------------- *)
(*--------------------------------- Fault Diagnosis and Management  ----------------------------------------------------- *)
(*----------------------------------------------------------------------------------------------------------------------- *)
(*Messaging*)
fB_MsgHandler();

IF eI_ELmodule_State = eFault THEN
  fB_Msg[1].bI_Status := TRUE;
ELSE
  fB_Msg[1].bI_Status := FALSE;
END_IF;
fB_Msg[1]();

fB_MsgQueue();


IF (bI_AckFault OR sI_CleanDevCmd.bAckError) AND NOT bL_memAckFault THEN
	tL_TimerSurv.IN:= FALSE;
END_IF;

IF bI_AckFault (*OR fb_MsgQueue.bO_ReceiptMessage*) OR sI_CleanDevCmd.bAckError THEN
	wL_ErrorCode := 0;
END_IF;

(*IF fL_diffDelta > 10000*iL_Precision THEN
	wL_ErrorCode.1 := TRUE;						(* Resolver Fault : delta is too large *)
END_IF;*)
wL_ErrorCode.1 := FALSE;
(*
IF fI_CurrentPosition < -(0.600) THEN	(*@@@@@@@@@@@@@ CONSTANT VALUE*)
	wL_ErrorCode.2:=TRUE;							(* Sensor Fault : Ref Sensor Expected *)
END_IF; *)

IF bL_MotionActive AND tL_TimerSurv.Q AND (fL_memX_Position = fI_CurrentPosition)  THEN			(* Motorization Fault, Command is active but position is not changing *)
	wL_ErrorCode.3 := TRUE;
END_IF;

IF (sI_SpeedDef_X.fP_PlaceSpeed = 0) OR (sI_SpeedDef_X.fP_WorkSpeed = 0) OR (sI_SpeedDef_X.fP_ServiceSpeed = 0) THEN	(* Speed Configuration not done *)
	wL_Errorcode.4 := TRUE;
END_IF;

IF (fI_CappPurgPosition=0) OR (fI_CleanRowPositions[1] = 0) THEN		(* Position Configuration not done *)
	wL_ErrorCode.5 := TRUE;
END_IF;

IF (eI_ELmodule_State = eFault) OR NOT bI_DeviceOnline THEN
	wL_ErrorCode.6 := TRUE;						(* EL7201 module fault *)
END_IF;

(*
IF bI_SafetyOk=FALSE AND bL_mem_SafetyOk=TRUE  THEN
	wL_ErrorCode.14:=TRUE;						(* Safety Fault *)
END_IF;*)

(*IF eI_ELmodule_State=eEstopped THEN
	wL_ErrorCode.15 :=TRUE;						(* EL7201 Emergency Stop*)
END_IF;*)
bL_mem_MoveEnable   := bO_MoveEnable;
bL_mem_MotionActive := bL_MotionActive;
bL_memAckFault      := bI_AckFault (*OR fb_MsgQueue.bO_ReceiptMessage*) OR sI_CleanDevCmd.bAckError;

bO_PositionUnknown  := NOT bL_Ref_Known;

ACTION Init:
	(*Messages*)
	sL_MsgConfig.bI_Enable       := TRUE;
	sL_MsgConfig.pI_FbMsgHandler := ADR(fB_MsgHandler);
	fB_MsgHandler.pI_MsgQueue    := ADR(fB_MsgQueue);
	fB_MsgQueue.pI_MsgInterface  := pC_MsgInterface;
	fB_MsgQueue.cI_MaxElement    := 5;

	fB_Msg[1].iI_MsgLocation     := iC_BlockId;
	fB_Msg[1].pI_MsgConfig       := ADR(sL_MsgConfig);
	fB_Msg[1].iI_MsgNumber       := eCMa_AxisErrorX;
END_ACTION

ACTION ProductionMode:
		bL_MotionActive:=FALSE;													(* stop when reach the RuhePosition*)
		bL_PrintReady	 :=TRUE;														(**)
		bL_AxisReady	 :=TRUE;
END_ACTION

ACTION ServiceMode:
(*Default speed*)
fO_SpeedLimit := sI_SpeedDef_X.fP_ServiceSpeed;

(*Mode selection*)
IF sI_CleanDevCmd.bAuto THEN	(*Control by cleaning process*)
	CASE 	sI_CleanDevCmd.eOperation OF
		eNOP:	(*No operation active*)
			bL_MotionActive:=FALSE;
			bL_AxisReady:=TRUE;
			bL_AfterHoming:=FALSE;

		eOPPREPSERVICE: (*Prepare service mode ---------------------------*)
			IF bL_AfterHoming THEN
				IF sI_CleanDevCmd.bInit THEN
					bL_MotionActive:=FALSE;
					bL_AxisReady:=TRUE;

				ELSIF sI_CleanDevCmd.bPrep THEN
					fO_TargetPosition :=fI_CappPurgPosition;
					bL_MotionActive:=TRUE;
					bL_AxisReady:=FALSE;
	
				ELSIF sI_CleanDevCmd.bStart THEN
					bL_MotionActive:=FALSE;
					bL_AxisReady:=TRUE;
	
				ELSIF sI_CleanDevCmd.bStop THEN
					bL_MotionActive:=FALSE;
					bL_AxisReady:=TRUE;
	
				ELSE	(*Command removed, wait until axis finished movement*)
					IF bL_MoveDone = FALSE THEN
						bL_MotionActive:=TRUE;
						bL_AxisReady:=FALSE;
					ELSE
						bL_MotionActive:=FALSE;
						bL_AxisReady:=TRUE;
					END_IF;
				END_IF;
			ELSE
				bL_MotionActive:=FALSE;
				bL_AxisReady:=TRUE;
			END_IF;

		eOPENDSERVICE: (*End service mode ---------------------------*)
			IF sI_CleanDevCmd.bInit THEN
				bL_MotionActive:=FALSE;
				bL_AxisReady:=TRUE;

			ELSIF sI_CleanDevCmd.bPrep THEN
				fO_TargetPosition :=fI_ParkPosition;
				bL_MotionActive:=TRUE;
				bL_AxisReady:=FALSE;

			ELSIF sI_CleanDevCmd.bStart THEN
				bL_MotionActive:=FALSE;
				bL_AxisReady:=TRUE;

			ELSIF sI_CleanDevCmd.bStop THEN
				bL_MotionActive:=FALSE;
				bL_AxisReady:=TRUE;

			ELSE	(*Command removed, wait until axis finished movement*)
				IF bL_MoveDone = FALSE THEN
					bL_MotionActive:=TRUE;
					bL_AxisReady:=FALSE;
				ELSE
					bL_MotionActive:=FALSE;
					bL_AxisReady:=TRUE;
				END_IF;
			END_IF;

		eOPCLEAN:	(*Cleaning Mode -------------------------------------*)
			IF sI_CleanDevCmd.bInit THEN
				fO_TargetPosition :=fI_CleanRowPositions[iI_CurrentCleanPos];
				bL_MotionActive:=TRUE;
				bL_AxisReady:=FALSE;

			ELSIF sI_CleanDevCmd.bPrep THEN
				fO_TargetPosition :=fI_CleanRowPositions[iI_CurrentCleanPos];
				bL_MotionActive:=FALSE;
				bL_AxisReady:=FALSE;

			ELSIF sI_CleanDevCmd.bStart THEN
				fO_TargetPosition :=fI_CleanRowPositions[iI_CurrentCleanPos];
				bL_MotionActive:=FALSE;
				bL_AxisReady:=FALSE;

			ELSIF sI_CleanDevCmd.bStop THEN
				fO_TargetPosition :=fI_CleanRowPositions[iI_CurrentCleanPos];
				bL_MotionActive:=FALSE;
				bL_AxisReady:=FALSE;

			ELSE	(*Command removed, wait until axis finished movement*)
				IF bL_MoveDone = FALSE THEN
					bL_MotionActive:=TRUE;
					bL_AxisReady:=FALSE;
				ELSE
					bL_MotionActive:=FALSE;
					bL_AxisReady:=TRUE;
				END_IF;
			END_IF;

		eOPPURGE:	(*Purge Mode -------------------------------------*)
			IF sI_CleanDevCmd.bInit THEN
				fO_TargetPosition :=fI_CappPurgPosition;
				bL_MotionActive:=TRUE;
				bL_AxisReady:=FALSE;

			ELSIF sI_CleanDevCmd.bPrep THEN
				fO_TargetPosition :=fI_CappPurgPosition;
				bL_MotionActive:=FALSE;
				bL_AxisReady:=FALSE;

			ELSIF sI_CleanDevCmd.bStart THEN
				fO_TargetPosition :=fI_CappPurgPosition;
				bL_MotionActive:=FALSE;
				bL_AxisReady:=FALSE;

			ELSIF sI_CleanDevCmd.bStop THEN
				fO_TargetPosition :=fI_CappPurgPosition;
				bL_MotionActive:=FALSE;
				bL_AxisReady:=FALSE;

			ELSE	(*Command removed, wait until axis finished movement*)
				IF bL_MoveDone = FALSE THEN
					bL_MotionActive:=TRUE;
					bL_AxisReady:=FALSE;
				ELSE
					bL_MotionActive:=FALSE;
					bL_AxisReady:=TRUE;
				END_IF;
			END_IF;

		eOPCAPENTER:	(*Enter Capping Mode -------------------------------------*)
			IF sI_CleanDevCmd.bInit THEN
				fO_TargetPosition :=fI_CappPurgPosition;
				bL_MotionActive:=TRUE;
				bL_AxisReady:=FALSE;

			ELSIF sI_CleanDevCmd.bPrep THEN
				fO_TargetPosition :=fI_CappPurgPosition;
				bL_MotionActive:=FALSE;
				bL_AxisReady:=FALSE;

			ELSIF sI_CleanDevCmd.bStart THEN
				fO_TargetPosition :=fI_CappPurgPosition;
				bL_MotionActive:=FALSE;
				bL_AxisReady:=FALSE;

			ELSIF sI_CleanDevCmd.bStop THEN
				fO_TargetPosition :=fI_CappPurgPosition;
				bL_MotionActive:=FALSE;
				bL_AxisReady:=FALSE;

			ELSE	(*Command removed, wait until axis finished movement*)
				IF bL_MoveDone = FALSE THEN
					bL_MotionActive:=TRUE;
					bL_AxisReady:=FALSE;
				ELSE
					bL_MotionActive:=FALSE;
					bL_AxisReady:=TRUE;
				END_IF;
			END_IF;

		eOPCAPEXIT:	(*Exit Capping Mode -------------------------------------*)
			IF sI_CleanDevCmd.bInit THEN
				fO_TargetPosition :=fI_CappPurgPosition;
				bL_MotionActive:=TRUE;
				bL_AxisReady:=FALSE;

			ELSIF sI_CleanDevCmd.bPrep THEN
				fO_TargetPosition :=fI_CappPurgPosition;
				bL_MotionActive:=TRUE;
				bL_AxisReady:=FALSE;

			ELSIF sI_CleanDevCmd.bStart THEN
				fO_TargetPosition :=fI_CappPurgPosition;
				bL_MotionActive:=TRUE;
				bL_AxisReady:=FALSE;

			ELSIF sI_CleanDevCmd.bStop THEN
				fO_TargetPosition :=fI_CappPurgPosition;
				bL_MotionActive:=TRUE;
				bL_AxisReady:=FALSE;

			ELSE	(*Command removed, wait until axis finished movement*)
				IF bL_MoveDone = FALSE THEN
					bL_MotionActive:=TRUE;
					bL_AxisReady:=FALSE;
				ELSE
					bL_MotionActive:=FALSE;
					bL_AxisReady:=TRUE;
				END_IF;
			END_IF;

		eOPMAINT:	(*Maintenance -------------------------------------*)
			IF sI_CleanDevCmd.bInit THEN
				fO_TargetPosition :=fI_ParkPosition;
				bL_MotionActive:=TRUE;
				bL_AxisReady:=FALSE;

			ELSIF sI_CleanDevCmd.bPrep THEN
				bL_MotionActive:=FALSE;
				bL_AxisReady:=TRUE;

			ELSIF sI_CleanDevCmd.bStart THEN
				bL_MotionActive:=FALSE;
				bL_AxisReady:=TRUE;

			ELSIF sI_CleanDevCmd.bStop THEN
				bL_MotionActive:=FALSE;
				bL_AxisReady:=TRUE;

			ELSE	(*Command removed, wait until axis finished movement*)
				IF bL_MoveDone = FALSE THEN
					bL_MotionActive:=TRUE;
					bL_AxisReady:=FALSE;
				ELSE
					bL_MotionActive:=FALSE;
					bL_AxisReady:=TRUE;
				END_IF;
			END_IF;
		eOPSHUTTEROPEN: (*Open Shutters, do nothing*)
			bL_AxisReady 			:= TRUE;
			bL_MotionActive		:= FALSE;

		ELSE
			bL_MotionActive:=FALSE;
			bL_AxisReady:=TRUE;
		END_CASE;

		(*In case of abort set target position to current position and wait for MoveDone flag*)
		IF sI_CleanDevCmd.bAbort THEN
			fO_TargetPosition := fI_CurrentPosition;
		END_IF;

ELSE		(* MANUAL MODE *)
	IF sI_ManualCommands.bI_Do=TRUE AND sI_ManualCommands.bI_Undo =FALSE THEN
		fO_TargetPosition := sI_ManualCommands.fI_Start_position ;
		bL_AxisReady:=FALSE;
	ELSIF sI_ManualCommands.bI_Do=FALSE AND sI_ManualCommands.bI_Undo =TRUE THEN
		fO_TargetPosition :=  sI_ManualCommands.fI_Stop_position;
		bL_AxisReady:=FALSE;
	ELSE
		fO_TargetPosition := fI_CurrentPosition;
		bL_AxisReady:=TRUE;
	END_IF;
	bL_MotionActive:=sI_ManualCommands.bI_Do OR sI_ManualCommands.bI_Undo;
END_IF;
END_ACTION

END_FUNCTION_BLOCK

// ---- POUs/Machine/CleaningStation/FB_EL7041.TcPOU
FUNCTION_BLOCK FB_EL7041
(*************************************************************************************************)
(*  FILENAME:    FB_EL7041                                                                       *)
(*  PROJECT:     CALMAR PUPLC                                                                    *)
(*  COPYRIGHT:   All rights reserved (c) Wifag//Polytype, Fribourg/Switzerland (2020)            *)
(*  ENVIRONMENT: TwinCAT PLC                                                                     *)
(*  VERSION:     <version>                                                                       *)
(*************************************************************************************************)
(*  DESCRIPTION:                                                                   <description> *)
(*    This function transfers the movement commands to the motor.                                *)
(*                                                                                </description> *)
(*************************************************************************************************)

{library PUBLIC}
VAR_INPUT
  fI_TargetPosition              : REAL;                         (*Target position [m]*)
  fI_Tolerance                   : REAL := 0.0001;               (*Position tolerance [m]*)
  fI_SpeedLimit                  : REAL;                         (*Speed limit [m/s]*)
  bI_MoveEnable                  : BOOL;                         (*Enable movement*)
  bI_RegActive                   : BOOL;                         (*Regulation active*)
  bI_FaultReset                  : BOOL;                         (*Fault reset*)
  bI_EStop                       : BOOL;                         (*Emergency stop*)
  bI_SetPosition                 : BOOL;                         (*Set position*)

  lI_EncoderValue                : DINT;                         (*Encoder value*)
  fI_Microstepping               : REAL := 64;                   (*Microstepping*)
  fI_LimitSpeedFullStep          : REAL := 37_500;               (*Limitb speed full step [U/m]*)
  fI_PosControllerGain           : REAL := 10.0;                 (*Position controller gain*)
  fI_EncoderScaling              : REAL := 12_800;               (*Encoder scaling [counts/rev]*)
  fI_Axis_Scaling                : REAL := 0.00125;              (*Axis scaling [m/rev]*)
  fI_SetPositionValue            : REAL := -0.001;               (*Set position value [m]*)
  //fI_SpeedScaling                : REAL := 500;                  (*Speed scaling [counts/rev]*)
END_VAR

VAR_OUTPUT
  iO_TargetVelocity              : DINT;                         (*Target velocity: 7010:21*)
  fO_ActualPosition              : REAL;                         (*Actual position [m]*)
  bO_MoveOk                      : BOOL;                         (*Movement ok*)
  bO_Error                       : BOOL;                         (*Modul error*)
END_VAR

{library private}
VAR
  fL_Delta_P                     : REAL;                         (*Delta position*)
  fL_CommandSignal               : REAL;                         (*Command signal*)

  tL_TimerRampUP                 : TON;                          (*Timer ramp up*)
  fL_PercentageRampUP            : REAL;                         (*Percentage ramp up*)
  tL_TimerRampDN                 : TON;                          (*Timer ramp down*)
  fL_PercentageRampDN            : REAL;                         (*Percentage ramp down*)

  bL_memMoveEnable               : BOOL;                         (*Memory enable movement*)
  bL_memSetPosition              : BOOL;                         (*Memory set position*)
  fL_memTargetPosition           : REAL := 0.0;                  (*Memory target position*)
  bL_StopRamp                    : BOOL;                         (*Stop ramp*)
  bL_FirstRun                    : BOOL := TRUE;                 (*First run*)

  fL_Divider                     : REAL;                         (*Divider for percent calculation*)
END_VAR

VAR PERSISTENT
  fL_OffsetEncoder               : DINT;                         (*Offset encoder*)
END_VAR

//Read inputs
Input();

tL_TimerRampUP.PT := T#300MS;
tL_TimerRampUP();

tL_TimerRampDN.PT := T#300MS;
tL_TimerRampDN();

IF NOT bI_MoveEnable AND bL_memMoveEnable THEN
  bL_StopRamp := TRUE;
END_IF;

IF bI_MoveEnable AND NOT bL_memMoveEnable THEN
  fL_memTargetPosition := fI_TargetPosition;
  bO_MoveOK            := FALSE;
ELSIF bL_FirstRun THEN
  fL_memTargetPosition := fO_ActualPosition;
END_IF;

IF tL_TimerRampDN.Q THEN
  bL_StopRamp := FALSE;
END_IF;

tL_TimerRampDN.IN := bL_StopRamp;

fL_Divider := TIME_TO_REAL(tL_TimerRampDN.PT);
IF fL_Divider <> 0 THEN
  fL_PercentageRampDN := TIME_TO_REAL(tL_TimerRampDN.ET) / fL_Divider;
END_IF;

tL_TimerRampUP.IN := bI_MoveEnable AND bI_RegActive;

fL_Divider := TIME_TO_REAL(tL_TimerRampUP.PT);
IF fL_Divider <> 0 THEN
  fL_PercentageRampUP := TIME_TO_REAL(tL_TimerRampUP.ET) / fL_Divider;
END_IF;

(* ---------------------- Calculation of the delta between the trget and the actual position -----------------*)
fL_Delta_P := fI_TargetPosition - fO_ActualPosition;

(* ---------------------- Calculation of the command signal for the target velocity  -------------------------*)
fL_CommandSignal := fL_Delta_P * fI_PosControllerGain;

